KUKA KRL program: EPS_2_251078_MH1A_A_20250930064554.src

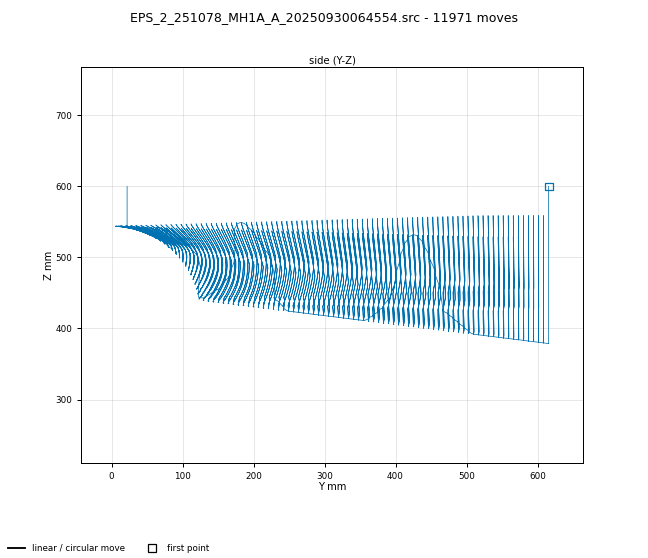
[picture p0: tool path of EPS_2_251078_MH1A_A_20250930064554.src, 11971 of 11973 moves have a stored position in this frame; points joined in program order, loops and branches not executed]
&ACCESS RVP
&REL 4
&COMMENT QRS 19112012
&PARAM EDITMASK = *
DEF PART()
EXT BAS (BAS_COMMAND :IN,REAL :IN )
INT I
BAS (#INITMOV,0 )

;KUKA QRS Post kuka4.cps  Date:22-06-2017 !

File_ID=2857

QRS_PRE_INIT()

;Init var - Until changes are made in qrs_pre_init
Outlet_Square_prg=0
Inlet_1_Square_prg=0
Inlet_2_Square_prg=0
Inlet_3_Square_prg=0
Inlet_4_Square_prg=0
Inlet_5_Square_prg=0

Outlet_1={X 0.000, Y 520.860, Z 458.500, B 0.000, E1 0.000 }
Inlet_1={X 0.000, Y 523.030, Z 428.500, B 0.000, E1 180.000 }
Outlet_1_type=201
Inlet_1_type=201
;QRS#1=Sidecore dimensions
;QRS#2=200-8" PVC SDR 35
;QRS#3=200-8" PVC SDR 35
;QRS#4=
;QRS#5=
;QRS#6=
;QRS#7=
;QRS#8=
;QRS#9=12-08 PSX
;QRS#10=12-08 PSX
;QRS#11=
;QRS#12=
;QRS#13=
;QRS#14=
;QRS#15=
;QRS#16=1220x127x838 2,75'
;QRS#17=EPS Height
;QRS#18=559
;QRS#19=*
;QRS#20= UPDATED VERSION 22-06-2017
;QRS#21=*
Outlet_Square=0100
Inlet_1_Square=0100
Inlet_2_Square=0
Inlet_3_Square=0
Inlet_4_Square=0
Inlet_5_Square=0
Mill_Square=1
Outlet_Square_Prg=204
Inlet_1_Square_prg=204

QRS_INIT()

$ADVANCE=5

; T1
PTP {E1 173.607,E2 173.607}
PTP {X 0,Y 615.504,A -85,B 0,C 180,E1 173.607,E2 173.607,E3 0,E4 0,E5 0,E6 0}
QRS_SPEED_INIT()
LIN {X 0,Y 615.504,Z 600,A -85,B 0,C 180,E1 173.607,E2 173.607,E3 0,E4 0,E5 0,E6 0} C_VEL
LIN {X 0,Y 615.504,Z 388.868,A -85,B 0,C 180,E1 173.607,E2 173.607} C_VEL
LIN {X 0,Y 615.504,Z 380.694,A -85,B 0,C 180,E1 173.607,E2 173.607} C_VEL
LIN {X 0,Y 615.49,Z 378.694,A -85,B 0,C 180,E1 173.421,E2 173.421} C_VEL
LIN {X 0,Y 615.492,Z 378.688,A -85,B 0,C 180,E1 170.801,E2 170.801} C_VEL
LIN {X 0,Y 615.493,Z 378.697,A -85,B 0,C 180,E1 168.139,E2 168.139} C_VEL
LIN {X 0,Y 615.481,Z 378.689,A -85,B 0,C 180,E1 165.451,E2 165.451} C_VEL
LIN {X 0,Y 615.492,Z 378.698,A -85,B 0,C 180,E1 162.73,E2 162.73} C_VEL
LIN {X 0,Y 615.49,Z 378.689,A -85,B 0,C 180,E1 159.967,E2 159.967} C_VEL
LIN {X 0,Y 615.486,Z 378.69,A -85,B 0,C 180,E1 157.155,E2 157.155} C_VEL
LIN {X 0,Y 615.5,Z 378.7,A -85,B 0,C 180,E1 154.285,E2 154.285} C_VEL
LIN {X 0,Y 615.478,Z 378.69,A -85,B 0,C 180,E1 151.552,E2 151.552} C_VEL
LIN {X 0,Y 615.487,Z 378.696,A -85,B 0,C 180,E1 148.914,E2 148.914} C_VEL
LIN {X 0,Y 615.489,Z 378.694,A -85,B 0,C 180,E1 145.978,E2 145.978} C_VEL
LIN {X 0,Y 615.487,Z 378.688,A -85,B 0,C 180,E1 143.064,E2 143.064} C_VEL
LIN {X 0,Y 615.49,Z 378.693,A -85,B 0,C 180,E1 140.25,E2 140.25} C_VEL
LIN {X 0,Y 615.477,Z 378.692,A -85,B 0,C 180,E1 137.646,E2 137.646} C_VEL
LIN {X 0,Y 615.48,Z 378.692,A -85,B 0,C 180,E1 134.93,E2 134.93} C_VEL
LIN {X 0,Y 615.49,Z 378.7,A -85,B 0,C 180,E1 132.08,E2 132.08} C_VEL
LIN {X 0,Y 615.479,Z 378.691,A -85,B 0,C 180,E1 129.751,E2 129.751} C_VEL
LIN {X 0,Y 615.488,Z 378.7,A -85,B 0,C 180,E1 126.936,E2 126.936} C_VEL
LIN {X 0,Y 615.485,Z 378.691,A -85,B 0,C 180,E1 125.616,E2 125.616} C_VEL
LIN {X 0,Y 615.482,Z 379.783,A -85,B 0,C 180,E1 124.699,E2 124.699} C_VEL
LIN {X 0,Y 615.494,Z 383.903,A -85,B 0,C 180,E1 122.331,E2 122.331} C_VEL
LIN {X 0,Y 615.496,Z 389.153,A -85,B 0,C 180,E1 119.406,E2 119.406} C_VEL
LIN {X 0,Y 615.486,Z 394.642,A -85,B 0,C 180,E1 116.444,E2 116.444} C_VEL
LIN {X 0,Y 615.49,Z 400.151,A -85,B 0,C 180,E1 113.556,E2 113.556} C_VEL
LIN {X 0,Y 615.487,Z 405.633,A -85,B 0,C 180,E1 110.731,E2 110.731} C_VEL
LIN {X 0,Y 615.483,Z 411.136,A -85,B 0,C 180,E1 107.957,E2 107.957} C_VEL
LIN {X 0,Y 615.484,Z 416.622,A -85,B 0,C 180,E1 105.226,E2 105.226} C_VEL
LIN {X 0,Y 615.483,Z 422.111,A -85,B 0,C 180,E1 102.53,E2 102.53} C_VEL
LIN {X 0,Y 615.492,Z 424.087,A -85,B 0,C 180,E1 101.568,E2 101.568} C_VEL
LIN {X 0,Y 615.484,Z 438.741,A -85,B 0,C 180,E1 101.235,E2 101.235} C_VEL
LIN {X 0,Y 615.491,Z 450.62,A -85,B 0,C 180,E1 100.842,E2 100.842} C_VEL
LIN {X 0,Y 615.478,Z 461.568,A -85,B 0,C 180,E1 100.361,E2 100.361} C_VEL
LIN {X 0,Y 615.497,Z 473.304,A -85,B 0,C 180,E1 99.696,E2 99.696} C_VEL
LIN {X 0,Y 615.499,Z 483.768,A -85,B 0,C 180,E1 98.95,E2 98.95} C_VEL
LIN {X 0,Y 615.498,Z 492.331,A -85,B 0,C 180,E1 98.206,E2 98.206} C_VEL
LIN {X 0,Y 615.497,Z 500.21,A -85,B 0,C 180,E1 97.38,E2 97.38} C_VEL
LIN {X 0,Y 615.497,Z 507.899,A -85,B 0,C 180,E1 96.392,E2 96.392} C_VEL
LIN {X 0,Y 615.497,Z 514.958,A -85,B 0,C 180,E1 95.241,E2 95.241} C_VEL
LIN {X 0,Y 615.494,Z 519.658,A -85,B 0,C 180,E1 94.256,E2 94.256} C_VEL
LIN {X 0,Y 615.494,Z 523.255,A -85,B 0,C 180,E1 93.273,E2 93.273} C_VEL
LIN {X 0,Y 615.496,Z 525.115,A -85,B 0,C 180,E1 92.618,E2 92.618} C_VEL
LIN {X 0,Y 615.5,Z 526.533,A -85,B 0,C 180,E1 91.963,E2 91.963} C_VEL
LIN {X 0,Y 615.496,Z 528.142,A -85,B 0,C 180,E1 90.654,E2 90.654} C_VEL
LIN {X 0,Y 615.495,Z 528.384,A -85,B 0,C 180,E1 90,E2 90} C_VEL
LIN {X 0,Y 615.495,Z 528.206,A -85,B 0,C 180,E1 89.346,E2 89.346} C_VEL
LIN {X 0,Y 615.5,Z 526.682,A -85,B 0,C 180,E1 88.037,E2 88.037} C_VEL
LIN {X 0,Y 615.498,Z 525.341,A -85,B 0,C 180,E1 87.382,E2 87.382} C_VEL
LIN {X 0,Y 615.496,Z 522.494,A -85,B 0,C 180,E1 86.399,E2 86.399} C_VEL
LIN {X 0,Y 615.498,Z 518.634,A -85,B 0,C 180,E1 85.415,E2 85.415} C_VEL
LIN {X 0,Y 615.498,Z 513.651,A -85,B 0,C 180,E1 84.43,E2 84.43} C_VEL
LIN {X 0,Y 615.496,Z 507.208,A -85,B 0,C 180,E1 83.418,E2 83.418} C_VEL
LIN {X 0,Y 615.497,Z 499.536,A -85,B 0,C 180,E1 82.455,E2 82.455} C_VEL
LIN {X 0,Y 615.498,Z 489.758,A -85,B 0,C 180,E1 81.463,E2 81.463} C_VEL
LIN {X 0,Y 615.498,Z 479.491,A -85,B 0,C 180,E1 80.636,E2 80.636} C_VEL
LIN {X 0,Y 615.482,Z 467.93,A -85,B 0,C 180,E1 79.889,E2 79.889} C_VEL
LIN {X 0,Y 615.491,Z 456.089,A -85,B 0,C 180,E1 79.294,E2 79.294} C_VEL
LIN {X 0,Y 615.477,Z 443.158,A -85,B 0,C 180,E1 78.807,E2 78.807} C_VEL
LIN {X 0,Y 615.487,Z 430.554,A -85,B 0,C 180,E1 78.473,E2 78.473} C_VEL
LIN {X 0,Y 615.496,Z 424.099,A -85,B 0,C 180,E1 78.348,E2 78.348} C_VEL
LIN {X 0,Y 615.481,Z 418.176,A -85,B 0,C 180,E1 75.451,E2 75.451} C_VEL
LIN {X 0,Y 615.486,Z 412.683,A -85,B 0,C 180,E1 72.729,E2 72.729} C_VEL
LIN {X 0,Y 615.479,Z 407.193,A -85,B 0,C 180,E1 69.967,E2 69.967} C_VEL
LIN {X 0,Y 615.486,Z 401.687,A -85,B 0,C 180,E1 67.155,E2 67.155} C_VEL
LIN {X 0,Y 615.487,Z 396.196,A -85,B 0,C 180,E1 64.284,E2 64.284} C_VEL
LIN {X 0,Y 615.491,Z 391.067,A -85,B 0,C 180,E1 61.55,E2 61.55} C_VEL
LIN {X 0,Y 615.488,Z 386.262,A -85,B 0,C 180,E1 58.914,E2 58.914} C_VEL
LIN {X 0,Y 615.495,Z 381.958,A -85,B 0,C 180,E1 56.465,E2 56.465} C_VEL
LIN {X 0,Y 615.483,Z 379.738,A -85,B 0,C 180,E1 55.184,E2 55.184} C_VEL
LIN {X 0,Y 615.485,Z 378.693,A -85,B 0,C 180,E1 54.384,E2 54.384} C_VEL
LIN {X 0,Y 615.481,Z 378.69,A -85,B 0,C 180,E1 51.931,E2 51.931} C_VEL
LIN {X 0,Y 615.485,Z 378.696,A -85,B 0,C 180,E1 49.393,E2 49.393} C_VEL
LIN {X 0,Y 615.496,Z 378.687,A -85,B 0,C 180,E1 46.756,E2 46.756} C_VEL
LIN {X 0,Y 615.484,Z 378.691,A -85,B 0,C 180,E1 43.997,E2 43.997} C_VEL
LIN {X 0,Y 615.491,Z 378.701,A -85,B 0,C 180,E1 41.095,E2 41.095} C_VEL
LIN {X 0,Y 615.494,Z 378.69,A -85,B 0,C 180,E1 38.904,E2 38.904} C_VEL
LIN {X 0,Y 615.478,Z 378.692,A -85,B 0,C 180,E1 36.426,E2 36.426} C_VEL
LIN {X 0,Y 615.487,Z 378.697,A -85,B 0,C 180,E1 34.022,E2 34.022} C_VEL
LIN {X 0,Y 615.482,Z 378.689,A -85,B 0,C 180,E1 31.686,E2 31.686} C_VEL
LIN {X 0,Y 615.48,Z 378.695,A -85,B 0,C 180,E1 29.407,E2 29.407} C_VEL
LIN {X 0,Y 615.498,Z 378.691,A -85,B 0,C 180,E1 27.046,E2 27.046} C_VEL
LIN {X 0,Y 615.487,Z 378.693,A -85,B 0,C 180,E1 24.272,E2 24.272} C_VEL
LIN {X 0,Y 615.479,Z 378.689,A -85,B 0,C 180,E1 21.432,E2 21.432} C_VEL
LIN {X 0,Y 615.481,Z 378.698,A -85,B 0,C 180,E1 18.602,E2 18.602} C_VEL
LIN {X 0,Y 615.48,Z 378.691,A -85,B 0,C 180,E1 15.905,E2 15.905} C_VEL
LIN {X 0,Y 615.494,Z 378.689,A -85,B 0,C 180,E1 13.201,E2 13.201} C_VEL
LIN {X 0,Y 615.486,Z 378.695,A -85,B 0,C 180,E1 10.527,E2 10.527} C_VEL
LIN {X 0,Y 615.477,Z 378.691,A -85,B 0,C 180,E1 7.876,E2 7.876} C_VEL
LIN {X 0,Y 615.495,Z 378.697,A -85,B 0,C 180,E1 5.241,E2 5.241} C_VEL
LIN {X 0,Y 615.488,Z 378.688,A -85,B 0,C 180,E1 2.618,E2 2.618} C_VEL
LIN {X 0,Y 615.486,Z 378.702,A -85,B 0,C 180,E1 0,E2 0} C_VEL
LIN {X 0,Y 615.488,Z 378.687,A -85,B 0,C 180,E1 -2.618,E2 -2.618} C_VEL
LIN {X 0,Y 615.489,Z 378.7,A -85,B 0,C 180,E1 -5.241,E2 -5.241} C_VEL
LIN {X 0,Y 615.478,Z 378.69,A -85,B 0,C 180,E1 -7.876,E2 -7.876} C_VEL
LIN {X 0,Y 615.485,Z 378.697,A -85,B 0,C 180,E1 -10.527,E2 -10.527} C_VEL
LIN {X 0,Y 615.494,Z 378.688,A -85,B 0,C 180,E1 -13.201,E2 -13.201} C_VEL
LIN {X 0,Y 615.485,Z 378.691,A -85,B 0,C 180,E1 -15.905,E2 -15.905} C_VEL
LIN {X 0,Y 615.49,Z 378.695,A -85,B 0,C 180,E1 -18.646,E2 -18.646} C_VEL
LIN {X 0,Y 615.478,Z 378.69,A -85,B 0,C 180,E1 -21.432,E2 -21.432} C_VEL
LIN {X 0,Y 615.484,Z 378.696,A -85,B 0,C 180,E1 -24.272,E2 -24.272} C_VEL
LIN {X 0,Y 615.497,Z 378.69,A -85,B 0,C 180,E1 -27.046,E2 -27.046} C_VEL
LIN {X 0,Y 615.488,Z 378.688,A -85,B 0,C 180,E1 -29.794,E2 -29.794} C_VEL
LIN {X 0,Y 615.49,Z 378.698,A -85,B 0,C 180,E1 -32.457,E2 -32.457} C_VEL
LIN {X 0,Y 615.49,Z 378.689,A -85,B 0,C 180,E1 -34.815,E2 -34.815} C_VEL
LIN {X 0,Y 615.481,Z 378.692,A -85,B 0,C 180,E1 -37.243,E2 -37.243} C_VEL
LIN {X 0,Y 615.483,Z 378.689,A -85,B 0,C 180,E1 -40.088,E2 -40.088} C_VEL
LIN {X 0,Y 615.477,Z 378.692,A -85,B 0,C 180,E1 -42.354,E2 -42.354} C_VEL
LIN {X 0,Y 615.48,Z 378.692,A -85,B 0,C 180,E1 -45.069,E2 -45.069} C_VEL
LIN {X 0,Y 615.495,Z 378.699,A -85,B 0,C 180,E1 -47.919,E2 -47.919} C_VEL
LIN {X 0,Y 615.478,Z 378.692,A -85,B 0,C 180,E1 -50.249,E2 -50.249} C_VEL
LIN {X 0,Y 615.483,Z 378.702,A -85,B 0,C 180,E1 -53.064,E2 -53.064} C_VEL
LIN {X 0,Y 615.49,Z 378.789,A -85,B 0,C 180,E1 -54.585,E2 -54.585} C_VEL
LIN {X 0,Y 615.495,Z 387.112,A -85,B 0,C 180,E1 -57.543,E2 -57.543} C_VEL
LIN {X 0,Y 615.479,Z 394.86,A -85,B 0,C 180,E1 -60.207,E2 -60.207} C_VEL
LIN {X 0,Y 615.478,Z 403.061,A -85,B 0,C 180,E1 -62.957,E2 -62.957} C_VEL
LIN {X 0,Y 615.495,Z 411.522,A -85,B 0,C 180,E1 -65.728,E2 -65.728} C_VEL
LIN {X 0,Y 615.485,Z 420.39,A -85,B 0,C 180,E1 -68.568,E2 -68.568} C_VEL
LIN {X 0,Y 615.488,Z 429.381,A -85,B 0,C 180,E1 -71.396,E2 -71.396} C_VEL
LIN {X 0,Y 615.485,Z 438.108,A -85,B 0,C 180,E1 -74.095,E2 -74.095} C_VEL
LIN {X 0,Y 615.494,Z 446.951,A -85,B 0,C 180,E1 -76.799,E2 -76.799} C_VEL
LIN {X 0,Y 615.491,Z 452.137,A -85,B 0,C 180,E1 -78.369,E2 -78.369} C_VEL
LIN {X 0,Y 615.499,Z 465.817,A -85,B 0,C 180,E1 -78.64,E2 -78.64} C_VEL
LIN {X 0,Y 615.489,Z 478.534,A -85,B 0,C 180,E1 -79.036,E2 -79.036} C_VEL
LIN {X 0,Y 615.479,Z 490.765,A -85,B 0,C 180,E1 -79.556,E2 -79.556} C_VEL
LIN {X 0,Y 615.498,Z 501.385,A -85,B 0,C 180,E1 -80.138,E2 -80.138} C_VEL
LIN {X 0,Y 615.498,Z 512.23,A -85,B 0,C 180,E1 -80.884,E2 -80.884} C_VEL
LIN {X 0,Y 615.497,Z 522.811,A -85,B 0,C 180,E1 -81.794,E2 -81.794} C_VEL
LIN {X 0,Y 615.498,Z 530.605,A -85,B 0,C 180,E1 -82.619,E2 -82.619} C_VEL
LIN {X 0,Y 615.496,Z 538.202,A -85,B 0,C 180,E1 -83.608,E2 -83.608} C_VEL
LIN {X 0,Y 615.498,Z 545.204,A -85,B 0,C 180,E1 -84.759,E2 -84.759} C_VEL
LIN {X 0,Y 615.493,Z 549.851,A -85,B 0,C 180,E1 -85.744,E2 -85.744} C_VEL
LIN {X 0,Y 615.495,Z 553.398,A -85,B 0,C 180,E1 -86.727,E2 -86.727} C_VEL
LIN {X 0,Y 615.497,Z 555.233,A -85,B 0,C 180,E1 -87.382,E2 -87.382} C_VEL
LIN {X 0,Y 615.499,Z 556.607,A -85,B 0,C 180,E1 -88.037,E2 -88.037} C_VEL
LIN {X 0,Y 615.496,Z 558.173,A -85,B 0,C 180,E1 -89.346,E2 -89.346} C_VEL
LIN {X 0,Y 615.494,Z 558.389,A -85,B 0,C 180,E1 -90,E2 -90} C_VEL
LIN {X 0,Y 615.496,Z 557.58,A -85,B 0,C 180,E1 -91.309,E2 -91.309} C_VEL
LIN {X 0,Y 615.499,Z 556.608,A -85,B 0,C 180,E1 -91.963,E2 -91.963} C_VEL
LIN {X 0,Y 615.497,Z 555.233,A -85,B 0,C 180,E1 -92.618,E2 -92.618} C_VEL
LIN {X 0,Y 615.496,Z 552.35,A -85,B 0,C 180,E1 -93.601,E2 -93.601} C_VEL
LIN {X 0,Y 615.498,Z 548.442,A -85,B 0,C 180,E1 -94.584,E2 -94.584} C_VEL
LIN {X 0,Y 615.499,Z 543.405,A -85,B 0,C 180,E1 -95.57,E2 -95.57} C_VEL
LIN {X 0,Y 615.497,Z 536.869,A -85,B 0,C 180,E1 -96.583,E2 -96.583} C_VEL
LIN {X 0,Y 615.497,Z 529.133,A -85,B 0,C 180,E1 -97.545,E2 -97.545} C_VEL
LIN {X 0,Y 615.498,Z 521.045,A -85,B 0,C 180,E1 -98.371,E2 -98.371} C_VEL
LIN {X 0,Y 615.499,Z 511.168,A -85,B 0,C 180,E1 -99.199,E2 -99.199} C_VEL
LIN {X 0,Y 615.491,Z 499.981,A -85,B 0,C 180,E1 -99.945,E2 -99.945} C_VEL
LIN {X 0,Y 615.481,Z 489.024,A -85,B 0,C 180,E1 -100.527,E2 -100.527} C_VEL
LIN {X 0,Y 615.489,Z 476.47,A -85,B 0,C 180,E1 -101.041,E2 -101.041} C_VEL
LIN {X 0,Y 615.498,Z 464.064,A -85,B 0,C 180,E1 -101.401,E2 -101.401} C_VEL
LIN {X 0,Y 615.491,Z 452.138,A -85,B 0,C 180,E1 -101.631,E2 -101.631} C_VEL
LIN {X 0,Y 615.476,Z 443.545,A -85,B 0,C 180,E1 -104.24,E2 -104.24} C_VEL
LIN {X 0,Y 615.483,Z 434.783,A -85,B 0,C 180,E1 -106.928,E2 -106.928} C_VEL
LIN {X 0,Y 615.485,Z 425.928,A -85,B 0,C 180,E1 -109.685,E2 -109.685} C_VEL
LIN {X 0,Y 615.491,Z 417.513,A -85,B 0,C 180,E1 -112.346,E2 -112.346} C_VEL
LIN {X 0,Y 615.478,Z 409.309,A -85,B 0,C 180,E1 -114.992,E2 -114.992} C_VEL
LIN {X 0,Y 615.494,Z 401.542,A -85,B 0,C 180,E1 -117.545,E2 -117.545} C_VEL
LIN {X 0,Y 615.497,Z 392.668,A -85,B 0,C 180,E1 -120.539,E2 -120.539} C_VEL
LIN {X 0,Y 615.491,Z 384.883,A -85,B 0,C 180,E1 -123.236,E2 -123.236} C_VEL
LIN {X 0,Y 615.489,Z 378.692,A -85,B 0,C 180,E1 -125.515,E2 -125.515} C_VEL
LIN {X 0,Y 615.481,Z 378.691,A -85,B 0,C 180,E1 -128.069,E2 -128.069} C_VEL
LIN {X 0,Y 615.482,Z 378.695,A -85,B 0,C 180,E1 -130.607,E2 -130.607} C_VEL
LIN {X 0,Y 615.496,Z 378.688,A -85,B 0,C 180,E1 -133.244,E2 -133.244} C_VEL
LIN {X 0,Y 615.488,Z 378.689,A -85,B 0,C 180,E1 -136.003,E2 -136.003} C_VEL
LIN {X 0,Y 615.488,Z 378.702,A -85,B 0,C 180,E1 -138.906,E2 -138.906} C_VEL
LIN {X 0,Y 615.49,Z 378.689,A -85,B 0,C 180,E1 -141.096,E2 -141.096} C_VEL
LIN {X 0,Y 615.478,Z 378.693,A -85,B 0,C 180,E1 -143.574,E2 -143.574} C_VEL
LIN {X 0,Y 615.494,Z 378.694,A -85,B 0,C 180,E1 -145.978,E2 -145.978} C_VEL
LIN {X 0,Y 615.482,Z 378.689,A -85,B 0,C 180,E1 -148.314,E2 -148.314} C_VEL
LIN {X 0,Y 615.483,Z 378.696,A -85,B 0,C 180,E1 -150.593,E2 -150.593} C_VEL
LIN {X 0,Y 615.497,Z 378.69,A -85,B 0,C 180,E1 -152.953,E2 -152.953} C_VEL
LIN {X 0,Y 615.484,Z 378.695,A -85,B 0,C 180,E1 -155.728,E2 -155.728} C_VEL
LIN {X 0,Y 615.478,Z 378.689,A -85,B 0,C 180,E1 -158.568,E2 -158.568} C_VEL
LIN {X 0,Y 615.488,Z 378.695,A -85,B 0,C 180,E1 -161.396,E2 -161.396} C_VEL
LIN {X 0,Y 615.482,Z 378.692,A -85,B 0,C 180,E1 -164.095,E2 -164.095} C_VEL
LIN {X 0,Y 615.494,Z 378.689,A -85,B 0,C 180,E1 -166.799,E2 -166.799} C_VEL
LIN {X 0,Y 615.486,Z 378.696,A -85,B 0,C 180,E1 -169.473,E2 -169.473} C_VEL
LIN {X 0,Y 615.478,Z 378.69,A -85,B 0,C 180,E1 -172.124,E2 -172.124} C_VEL
LIN {X 0,Y 615.489,Z 378.699,A -85,B 0,C 180,E1 -174.759,E2 -174.759} C_VEL
LIN {X 0,Y 615.488,Z 378.687,A -85,B 0,C 180,E1 -177.382,E2 -177.382} C_VEL
LIN {X 0,Y 615.489,Z 378.702,A -85,B 0,C 180,E1 -180,E2 -180} C_VEL
LIN {X 0,Y 615.488,Z 378.687,A -85,B 0,C 180,E1 -182.618,E2 -182.618} C_VEL
LIN {X 0,Y 615.495,Z 378.698,A -85,B 0,C 180,E1 -185.241,E2 -185.241} C_VEL
LIN {X 0,Y 615.49,Z 378.694,A -85,B 0,C 180,E1 -186.579,E2 -186.579} C_VEL
LIN {X 0,Y 614.817,Z 378.84,A -85,B 0,C 180,E1 -187.125,E2 -187.125} C_VEL
LIN {X 0,Y 611.985,Z 379.251,A -85,B 0,C 180,E1 -188.011,E2 -188.011} C_VEL
LIN {X 0,Y 609.592,Z 379.56,A -85,B 0,C 180,E1 -188.724,E2 -188.724} C_VEL
LIN {X 0,Y 608.552,Z 379.679,A -85,B 0,C 180,E1 -189.273,E2 -189.273} C_VEL
LIN {X 0,Y 608.461,Z 379.689,A -85,B 0,C 180,E1 -189.459,E2 -189.459} C_VEL
LIN {X 0,Y 608.466,Z 379.697,A -85,B 0,C 180,E1 -192,E2 -192} C_VEL
LIN {X 0,Y 608.474,Z 379.688,A -85,B 0,C 180,E1 -194.721,E2 -194.721} C_VEL
LIN {X 0,Y 608.455,Z 379.693,A -85,B 0,C 180,E1 -197.477,E2 -197.477} C_VEL
LIN {X 0,Y 608.465,Z 379.692,A -85,B 0,C 180,E1 -200.274,E2 -200.274} C_VEL
LIN {X 0,Y 608.449,Z 379.691,A -85,B 0,C 180,E1 -203.124,E2 -203.124} C_VEL
LIN {X 0,Y 608.481,Z 379.695,A -85,B 0,C 180,E1 -205.722,E2 -205.722} C_VEL
LIN {X 0,Y 608.446,Z 379.691,A -85,B 0,C 180,E1 -208.267,E2 -208.267} C_VEL
LIN {X 0,Y 608.476,Z 379.69,A -85,B 0,C 180,E1 -210.545,E2 -210.545} C_VEL
LIN {X 0,Y 608.455,Z 379.693,A -85,B 0,C 180,E1 -212.88,E2 -212.88} C_VEL
LIN {X 0,Y 608.443,Z 379.691,A -85,B 0,C 180,E1 -215.278,E2 -215.278} C_VEL
LIN {X 0,Y 608.468,Z 379.696,A -85,B 0,C 180,E1 -217.747,E2 -217.747} C_VEL
LIN {X 0,Y 608.448,Z 379.691,A -85,B 0,C 180,E1 -220.328,E2 -220.328} C_VEL
LIN {X 0,Y 608.449,Z 379.697,A -85,B 0,C 180,E1 -222.96,E2 -222.96} C_VEL
LIN {X 0,Y 608.46,Z 379.69,A -85,B 0,C 180,E1 -225.736,E2 -225.736} C_VEL
LIN {X 0,Y 608.465,Z 379.689,A -85,B 0,C 180,E1 -228.658,E2 -228.658} C_VEL
LIN {X 0,Y 608.465,Z 379.692,A -85,B 0,C 180,E1 -231.76,E2 -231.76} C_VEL
LIN {X 0,Y 608.447,Z 379.691,A -85,B 0,C 180,E1 -233.955,E2 -233.955} C_VEL
LIN {X 0,Y 608.413,Z 379.769,A -85,B 0,C 180,E1 -234.72,E2 -234.72} C_VEL
LIN {X 0,Y 608.464,Z 383.894,A -85,B 0,C 180,E1 -237.121,E2 -237.121} C_VEL
LIN {X 0,Y 608.443,Z 389.024,A -85,B 0,C 180,E1 -240.033,E2 -240.033} C_VEL
LIN {X 0,Y 608.445,Z 394.097,A -85,B 0,C 180,E1 -242.799,E2 -242.799} C_VEL
LIN {X 0,Y 608.423,Z 399.036,A -85,B 0,C 180,E1 -245.428,E2 -245.428} C_VEL
LIN {X 0,Y 608.446,Z 404.566,A -85,B 0,C 180,E1 -248.308,E2 -248.308} C_VEL
LIN {X 0,Y 608.427,Z 410.427,A -85,B 0,C 180,E1 -251.297,E2 -251.297} C_VEL
LIN {X 0,Y 608.442,Z 415.625,A -85,B 0,C 180,E1 -253.906,E2 -253.906} C_VEL
LIN {X 0,Y 608.425,Z 421.155,A -85,B 0,C 180,E1 -256.643,E2 -256.643} C_VEL
LIN {X 0,Y 608.45,Z 424.524,A -85,B 0,C 180,E1 -258.296,E2 -258.296} C_VEL
LIN {X 0,Y 608.526,Z 440.394,A -85,B 0,C 180,E1 -258.677,E2 -258.677} C_VEL
LIN {X 0,Y 608.532,Z 452.792,A -85,B 0,C 180,E1 -259.113,E2 -259.113} C_VEL
LIN {X 0,Y 608.48,Z 464.935,A -85,B 0,C 180,E1 -259.687,E2 -259.687} C_VEL
LIN {X 0,Y 608.5,Z 476.067,A -85,B 0,C 180,E1 -260.359,E2 -260.359} C_VEL
LIN {X 0,Y 608.474,Z 485.084,A -85,B 0,C 180,E1 -261.029,E2 -261.029} C_VEL
LIN {X 0,Y 608.464,Z 494.35,A -85,B 0,C 180,E1 -261.866,E2 -261.866} C_VEL
LIN {X 0,Y 608.466,Z 503.324,A -85,B 0,C 180,E1 -262.867,E2 -262.867} C_VEL
LIN {X 0,Y 608.444,Z 510.556,A -85,B 0,C 180,E1 -263.867,E2 -263.867} C_VEL
LIN {X 0,Y 608.462,Z 515.435,A -85,B 0,C 180,E1 -264.698,E2 -264.698} C_VEL
LIN {X 0,Y 608.439,Z 520.178,A -85,B 0,C 180,E1 -265.694,E2 -265.694} C_VEL
LIN {X 0,Y 608.425,Z 523.812,A -85,B 0,C 180,E1 -266.689,E2 -266.689} C_VEL
LIN {X 0,Y 608.425,Z 525.691,A -85,B 0,C 180,E1 -267.352,E2 -267.352} C_VEL
LIN {X 0,Y 608.444,Z 527.127,A -85,B 0,C 180,E1 -268.014,E2 -268.014} C_VEL
LIN {X 0,Y 608.439,Z 528.752,A -85,B 0,C 180,E1 -269.338,E2 -269.338} C_VEL
LIN {X 0,Y 608.435,Z 528.995,A -85,B 0,C 180,E1 -270,E2 -270} C_VEL
LIN {X 0,Y 608.438,Z 528.815,A -85,B 0,C 180,E1 -270.662,E2 -270.662} C_VEL
LIN {X 0,Y 608.445,Z 527.276,A -85,B 0,C 180,E1 -271.986,E2 -271.986} C_VEL
LIN {X 0,Y 608.426,Z 525.918,A -85,B 0,C 180,E1 -272.648,E2 -272.648} C_VEL
LIN {X 0,Y 608.449,Z 523.041,A -85,B 0,C 180,E1 -273.642,E2 -273.642} C_VEL
LIN {X 0,Y 608.433,Z 519.142,A -85,B 0,C 180,E1 -274.638,E2 -274.638} C_VEL
LIN {X 0,Y 608.45,Z 514.112,A -85,B 0,C 180,E1 -275.634,E2 -275.634} C_VEL
LIN {X 0,Y 608.441,Z 507.794,A -85,B 0,C 180,E1 -276.633,E2 -276.633} C_VEL
LIN {X 0,Y 608.475,Z 499.878,A -85,B 0,C 180,E1 -277.633,E2 -277.633} C_VEL
LIN {X 0,Y 608.472,Z 490.035,A -85,B 0,C 180,E1 -278.636,E2 -278.636} C_VEL
LIN {X 0,Y 608.481,Z 479.712,A -85,B 0,C 180,E1 -279.473,E2 -279.473} C_VEL
LIN {X 0,Y 608.478,Z 468.098,A -85,B 0,C 180,E1 -280.229,E2 -280.229} C_VEL
LIN {X 0,Y 608.507,Z 456.22,A -85,B 0,C 180,E1 -280.831,E2 -280.831} C_VEL
LIN {X 0,Y 608.521,Z 443.258,A -85,B 0,C 180,E1 -281.323,E2 -281.323} C_VEL
LIN {X 0,Y 608.546,Z 430.64,A -85,B 0,C 180,E1 -281.66,E2 -281.66} C_VEL
LIN {X 0,Y 608.446,Z 424.535,A -85,B 0,C 180,E1 -281.789,E2 -281.789} C_VEL
LIN {X 0,Y 608.413,Z 418.571,A -85,B 0,C 180,E1 -284.722,E2 -284.722} C_VEL
LIN {X 0,Y 608.432,Z 413.039,A -85,B 0,C 180,E1 -287.477,E2 -287.477} C_VEL
LIN {X 0,Y 608.425,Z 407.506,A -85,B 0,C 180,E1 -290.276,E2 -290.276} C_VEL
LIN {X 0,Y 608.432,Z 403.236,A -85,B 0,C 180,E1 -292.469,E2 -292.469} C_VEL
LIN {X 0,Y 608.435,Z 397.824,A -85,B 0,C 180,E1 -295.302,E2 -295.302} C_VEL
LIN {X 0,Y 608.45,Z 393.674,A -85,B 0,C 180,E1 -297.518,E2 -297.518} C_VEL
LIN {X 0,Y 608.443,Z 389.187,A -85,B 0,C 180,E1 -299.967,E2 -299.967} C_VEL
LIN {X 0,Y 608.465,Z 384.028,A -85,B 0,C 180,E1 -302.879,E2 -302.879} C_VEL
LIN {X 0,Y 608.414,Z 379.924,A -85,B 0,C 180,E1 -305.28,E2 -305.28} C_VEL
LIN {X 0,Y 608.484,Z 379.691,A -85,B 0,C 180,E1 -307.16,E2 -307.16} C_VEL
LIN {X 0,Y 608.443,Z 379.691,A -85,B 0,C 180,E1 -309.442,E2 -309.442} C_VEL
LIN {X 0,Y 608.466,Z 379.693,A -85,B 0,C 180,E1 -312.334,E2 -312.334} C_VEL
LIN {X 0,Y 608.452,Z 379.69,A -85,B 0,C 180,E1 -314.797,E2 -314.797} C_VEL
LIN {X 0,Y 608.448,Z 379.696,A -85,B 0,C 180,E1 -317.039,E2 -317.039} C_VEL
LIN {X 0,Y 608.456,Z 379.69,A -85,B 0,C 180,E1 -319.697,E2 -319.697} C_VEL
LIN {X 0,Y 608.467,Z 379.695,A -85,B 0,C 180,E1 -322.253,E2 -322.253} C_VEL
LIN {X 0,Y 608.456,Z 379.69,A -85,B 0,C 180,E1 -325.094,E2 -325.094} C_VEL
LIN {X 0,Y 608.465,Z 379.691,A -85,B 0,C 180,E1 -327.905,E2 -327.905} C_VEL
LIN {X 0,Y 608.47,Z 379.688,A -85,B 0,C 180,E1 -330.22,E2 -330.22} C_VEL
LIN {X 0,Y 608.488,Z 379.691,A -85,B 0,C 180,E1 -332.791,E2 -332.791} C_VEL
LIN {X 0,Y 608.457,Z 379.69,A -85,B 0,C 180,E1 -335.429,E2 -335.429} C_VEL
LIN {X 0,Y 608.468,Z 379.689,A -85,B 0,C 180,E1 -338.308,E2 -338.308} C_VEL
LIN {X 0,Y 608.457,Z 379.697,A -85,B 0,C 180,E1 -341.13,E2 -341.13} C_VEL
LIN {X 0,Y 608.458,Z 379.69,A -85,B 0,C 180,E1 -343.906,E2 -343.906} C_VEL
LIN {X 0,Y 608.468,Z 379.692,A -85,B 0,C 180,E1 -346.644,E2 -346.644} C_VEL
LIN {X 0,Y 608.462,Z 379.691,A -85,B 0,C 180,E1 -349.35,E2 -349.35} C_VEL
LIN {X 0,Y 608.473,Z 379.689,A -85,B 0,C 180,E1 -352.033,E2 -352.033} C_VEL
LIN {X 0,Y 608.472,Z 379.693,A -85,B 0,C 180,E1 -354.698,E2 -354.698} C_VEL
LIN {X 0,Y 608.479,Z 379.687,A -85,B 0,C 180,E1 -357.352,E2 -357.352} C_VEL
LIN {X 0,Y 608.477,Z 379.695,A -85,B 0,C 180,E1 -360,E2 -360} C_VEL
LIN {X 0,Y 608.479,Z 379.687,A -85,B 0,C 180,E1 -362.648,E2 -362.648} C_VEL
LIN {X 0,Y 608.467,Z 379.694,A -85,B 0,C 180,E1 -365.302,E2 -365.302} C_VEL
LIN {X 0,Y 608.473,Z 379.688,A -85,B 0,C 180,E1 -367.967,E2 -367.967} C_VEL
LIN {X 0,Y 608.461,Z 379.692,A -85,B 0,C 180,E1 -370.65,E2 -370.65} C_VEL
LIN {X 0,Y 608.471,Z 379.69,A -85,B 0,C 180,E1 -373.356,E2 -373.356} C_VEL
LIN {X 0,Y 608.461,Z 379.69,A -85,B 0,C 180,E1 -376.094,E2 -376.094} C_VEL
LIN {X 0,Y 608.46,Z 379.697,A -85,B 0,C 180,E1 -378.87,E2 -378.87} C_VEL
LIN {X 0,Y 608.467,Z 379.689,A -85,B 0,C 180,E1 -381.692,E2 -381.692} C_VEL
LIN {X 0,Y 608.455,Z 379.691,A -85,B 0,C 180,E1 -384.571,E2 -384.571} C_VEL
LIN {X 0,Y 608.488,Z 379.69,A -85,B 0,C 180,E1 -387.208,E2 -387.208} C_VEL
LIN {X 0,Y 608.47,Z 379.688,A -85,B 0,C 180,E1 -389.971,E2 -389.971} C_VEL
LIN {X 0,Y 608.458,Z 379.693,A -85,B 0,C 180,E1 -392.88,E2 -392.88} C_VEL
LIN {X 0,Y 608.442,Z 379.692,A -85,B 0,C 180,E1 -395.278,E2 -395.278} C_VEL
LIN {X 0,Y 608.467,Z 379.696,A -85,B 0,C 180,E1 -397.747,E2 -397.747} C_VEL
LIN {X 0,Y 608.447,Z 379.691,A -85,B 0,C 180,E1 -400.328,E2 -400.328} C_VEL
LIN {X 0,Y 608.452,Z 379.697,A -85,B 0,C 180,E1 -402.96,E2 -402.96} C_VEL
LIN {X 0,Y 608.463,Z 379.69,A -85,B 0,C 180,E1 -405.736,E2 -405.736} C_VEL
LIN {X 0,Y 608.463,Z 379.689,A -85,B 0,C 180,E1 -408.658,E2 -408.658} C_VEL
LIN {X 0,Y 608.464,Z 379.692,A -85,B 0,C 180,E1 -411.76,E2 -411.76} C_VEL
LIN {X 0,Y 608.513,Z 379.891,A -85,B 0,C 180,E1 -414.524,E2 -414.524} C_VEL
LIN {X 0,Y 608.496,Z 388.146,A -85,B 0,C 180,E1 -417.473,E2 -417.473} C_VEL
LIN {X 0,Y 608.471,Z 396.073,A -85,B 0,C 180,E1 -420.22,E2 -420.22} C_VEL
LIN {X 0,Y 608.474,Z 403.68,A -85,B 0,C 180,E1 -422.794,E2 -422.794} C_VEL
LIN {X 0,Y 608.466,Z 411.656,A -85,B 0,C 180,E1 -425.429,E2 -425.429} C_VEL
LIN {X 0,Y 608.453,Z 420.56,A -85,B 0,C 180,E1 -428.308,E2 -428.308} C_VEL
LIN {X 0,Y 608.46,Z 429.465,A -85,B 0,C 180,E1 -431.13,E2 -431.13} C_VEL
LIN {X 0,Y 608.442,Z 438.369,A -85,B 0,C 180,E1 -433.906,E2 -433.906} C_VEL
LIN {X 0,Y 608.438,Z 447.274,A -85,B 0,C 180,E1 -436.643,E2 -436.643} C_VEL
LIN {X 0,Y 608.436,Z 452.491,A -85,B 0,C 180,E1 -438.232,E2 -438.232} C_VEL
LIN {X 0,Y 608.544,Z 466.693,A -85,B 0,C 180,E1 -438.53,E2 -438.53} C_VEL
LIN {X 0,Y 608.521,Z 479.464,A -85,B 0,C 180,E1 -438.939,E2 -438.939} C_VEL
LIN {X 0,Y 608.51,Z 490.919,A -85,B 0,C 180,E1 -439.435,E2 -439.435} C_VEL
LIN {X 0,Y 608.489,Z 501.577,A -85,B 0,C 180,E1 -440.023,E2 -440.023} C_VEL
LIN {X 0,Y 608.483,Z 512.473,A -85,B 0,C 180,E1 -440.778,E2 -440.778} C_VEL
LIN {X 0,Y 608.475,Z 523.111,A -85,B 0,C 180,E1 -441.699,E2 -441.699} C_VEL
LIN {X 0,Y 608.471,Z 530.959,A -85,B 0,C 180,E1 -442.534,E2 -442.534} C_VEL
LIN {X 0,Y 608.461,Z 538.286,A -85,B 0,C 180,E1 -443.484,E2 -443.484} C_VEL
LIN {X 0,Y 608.45,Z 543.865,A -85,B 0,C 180,E1 -444.366,E2 -444.366} C_VEL
LIN {X 0,Y 608.432,Z 548.95,A -85,B 0,C 180,E1 -445.362,E2 -445.362} C_VEL
LIN {X 0,Y 608.449,Z 552.896,A -85,B 0,C 180,E1 -446.358,E2 -446.358} C_VEL
LIN {X 0,Y 608.425,Z 555.809,A -85,B 0,C 180,E1 -447.352,E2 -447.352} C_VEL
LIN {X 0,Y 608.444,Z 557.201,A -85,B 0,C 180,E1 -448.014,E2 -448.014} C_VEL
LIN {X 0,Y 608.438,Z 558.783,A -85,B 0,C 180,E1 -449.338,E2 -449.338} C_VEL
LIN {X 0,Y 608.434,Z 559,A -85,B 0,C 180,E1 -450,E2 -450} C_VEL
LIN {X 0,Y 608.448,Z 558.184,A -85,B 0,C 180,E1 -451.324,E2 -451.324} C_VEL
LIN {X 0,Y 608.444,Z 557.201,A -85,B 0,C 180,E1 -451.986,E2 -451.986} C_VEL
LIN {X 0,Y 608.425,Z 555.809,A -85,B 0,C 180,E1 -452.648,E2 -452.648} C_VEL
LIN {X 0,Y 608.449,Z 552.896,A -85,B 0,C 180,E1 -453.642,E2 -453.642} C_VEL
LIN {X 0,Y 608.432,Z 548.95,A -85,B 0,C 180,E1 -454.638,E2 -454.638} C_VEL
LIN {X 0,Y 608.437,Z 542.877,A -85,B 0,C 180,E1 -455.801,E2 -455.801} C_VEL
LIN {X 0,Y 608.462,Z 536.235,A -85,B 0,C 180,E1 -456.799,E2 -456.799} C_VEL
LIN {X 0,Y 608.455,Z 527.989,A -85,B 0,C 180,E1 -457.8,E2 -457.8} C_VEL
LIN {X 0,Y 608.472,Z 519.537,A -85,B 0,C 180,E1 -458.636,E2 -458.636} C_VEL
LIN {X 0,Y 608.481,Z 509.091,A -85,B 0,C 180,E1 -459.473,E2 -459.473} C_VEL
LIN {X 0,Y 608.491,Z 498.756,A -85,B 0,C 180,E1 -460.145,E2 -460.145} C_VEL
LIN {X 0,Y 608.518,Z 487.26,A -85,B 0,C 180,E1 -460.74,E2 -460.74} C_VEL
LIN {X 0,Y 608.537,Z 474.892,A -85,B 0,C 180,E1 -461.224,E2 -461.224} C_VEL
LIN {X 0,Y 608.546,Z 461.44,A -85,B 0,C 180,E1 -461.597,E2 -461.597} C_VEL
LIN {X 0,Y 608.436,Z 452.492,A -85,B 0,C 180,E1 -461.768,E2 -461.768} C_VEL
LIN {X 0,Y 608.424,Z 443.935,A -85,B 0,C 180,E1 -464.38,E2 -464.38} C_VEL
LIN {X 0,Y 608.451,Z 436.144,A -85,B 0,C 180,E1 -466.784,E2 -466.784} C_VEL
LIN {X 0,Y 608.457,Z 427.239,A -85,B 0,C 180,E1 -469.57,E2 -469.57} C_VEL
LIN {X 0,Y 608.48,Z 418.335,A -85,B 0,C 180,E1 -472.405,E2 -472.405} C_VEL
LIN {X 0,Y 608.465,Z 410.543,A -85,B 0,C 180,E1 -474.935,E2 -474.935} C_VEL
LIN {X 0,Y 608.473,Z 402.752,A -85,B 0,C 180,E1 -477.517,E2 -477.517} C_VEL
LIN {X 0,Y 608.485,Z 395.504,A -85,B 0,C 180,E1 -479.974,E2 -479.974} C_VEL
LIN {X 0,Y 608.498,Z 387.146,A -85,B 0,C 180,E1 -482.877,E2 -482.877} C_VEL
LIN {X 0,Y 608.463,Z 379.692,A -85,B 0,C 180,E1 -485.581,E2 -485.581} C_VEL
LIN {X 0,Y 608.464,Z 379.692,A -85,B 0,C 180,E1 -488.24,E2 -488.24} C_VEL
LIN {X 0,Y 608.463,Z 379.689,A -85,B 0,C 180,E1 -491.342,E2 -491.342} C_VEL
LIN {X 0,Y 608.463,Z 379.69,A -85,B 0,C 180,E1 -494.264,E2 -494.264} C_VEL
LIN {X 0,Y 608.449,Z 379.697,A -85,B 0,C 180,E1 -497.04,E2 -497.04} C_VEL
LIN {X 0,Y 608.454,Z 379.69,A -85,B 0,C 180,E1 -499.697,E2 -499.697} C_VEL
LIN {X 0,Y 608.466,Z 379.696,A -85,B 0,C 180,E1 -502.253,E2 -502.253} C_VEL
LIN {X 0,Y 608.442,Z 379.692,A -85,B 0,C 180,E1 -504.722,E2 -504.722} C_VEL
LIN {X 0,Y 608.466,Z 379.696,A -85,B 0,C 180,E1 -507.477,E2 -507.477} C_VEL
LIN {X 0,Y 608.472,Z 379.688,A -85,B 0,C 180,E1 -510.221,E2 -510.221} C_VEL
LIN {X 0,Y 608.488,Z 379.69,A -85,B 0,C 180,E1 -512.791,E2 -512.791} C_VEL
LIN {X 0,Y 608.455,Z 379.691,A -85,B 0,C 180,E1 -515.429,E2 -515.429} C_VEL
LIN {X 0,Y 608.467,Z 379.689,A -85,B 0,C 180,E1 -518.308,E2 -518.308} C_VEL
LIN {X 0,Y 608.458,Z 379.697,A -85,B 0,C 180,E1 -521.13,E2 -521.13} C_VEL
LIN {X 0,Y 608.459,Z 379.69,A -85,B 0,C 180,E1 -523.906,E2 -523.906} C_VEL
LIN {X 0,Y 608.471,Z 379.691,A -85,B 0,C 180,E1 -526.644,E2 -526.644} C_VEL
LIN {X 0,Y 608.462,Z 379.692,A -85,B 0,C 180,E1 -529.35,E2 -529.35} C_VEL
LIN {X 0,Y 608.473,Z 379.688,A -85,B 0,C 180,E1 -532.033,E2 -532.033} C_VEL
LIN {X 0,Y 608.467,Z 379.694,A -85,B 0,C 180,E1 -534.698,E2 -534.698} C_VEL
LIN {X 0,Y 608.479,Z 379.687,A -85,B 0,C 180,E1 -537.352,E2 -537.352} C_VEL
LIN {X 0,Y 608.48,Z 379.695,A -85,B 0,C 180,E1 -540,E2 -540} C_VEL
LIN {X 0,Y 608.479,Z 379.687,A -85,B 0,C 180,E1 -542.648,E2 -542.648} C_VEL
LIN {X 0,Y 608.473,Z 379.693,A -85,B 0,C 180,E1 -545.302,E2 -545.302} C_VEL
LIN {X 0,Y 608.473,Z 379.688,A -85,B 0,C 180,E1 -547.967,E2 -547.967} C_VEL
LIN {X 0,Y 608.461,Z 379.689,A -85,B 0,C 180,E1 -549.459,E2 -549.459} C_VEL
LIN {X 0,Y 607.777,Z 379.779,A -85,B 0,C 180,E1 -550.012,E2 -550.012} C_VEL
LIN {X 0,Y 604.924,Z 380.136,A -85,B 0,C 180,E1 -550.909,E2 -550.909} C_VEL
LIN {X 0,Y 602.525,Z 380.436,A -85,B 0,C 180,E1 -551.63,E2 -551.63} C_VEL
LIN {X 0,Y 601.496,Z 380.562,A -85,B 0,C 180,E1 -552.187,E2 -552.187} C_VEL
LIN {X 0,Y 601.412,Z 380.57,A -85,B 0,C 180,E1 -552.376,E2 -552.376} C_VEL
LIN {X 0,Y 601.43,Z 380.566,A -85,B 0,C 180,E1 -554.897,E2 -554.897} C_VEL
LIN {X 0,Y 601.424,Z 380.571,A -85,B 0,C 180,E1 -556.986,E2 -556.986} C_VEL
LIN {X 0,Y 601.409,Z 380.568,A -85,B 0,C 180,E1 -559.809,E2 -559.809} C_VEL
LIN {X 0,Y 601.414,Z 380.569,A -85,B 0,C 180,E1 -562.683,E2 -562.683} C_VEL
LIN {X 0,Y 601.407,Z 380.568,A -85,B 0,C 180,E1 -564.879,E2 -564.879} C_VEL
LIN {X 0,Y 601.425,Z 380.573,A -85,B 0,C 180,E1 -567.364,E2 -567.364} C_VEL
LIN {X 0,Y 601.431,Z 380.565,A -85,B 0,C 180,E1 -570.164,E2 -570.164} C_VEL
LIN {X 0,Y 601.42,Z 380.572,A -85,B 0,C 180,E1 -572.715,E2 -572.715} C_VEL
LIN {X 0,Y 601.414,Z 380.567,A -85,B 0,C 180,E1 -575.114,E2 -575.114} C_VEL
LIN {X 0,Y 601.437,Z 380.568,A -85,B 0,C 180,E1 -577.419,E2 -577.419} C_VEL
LIN {X 0,Y 601.414,Z 380.568,A -85,B 0,C 180,E1 -579.995,E2 -579.995} C_VEL
LIN {X 0,Y 601.41,Z 380.573,A -85,B 0,C 180,E1 -582.671,E2 -582.671} C_VEL
LIN {X 0,Y 601.429,Z 380.565,A -85,B 0,C 180,E1 -585.482,E2 -585.482} C_VEL
LIN {X 0,Y 601.428,Z 380.568,A -85,B 0,C 180,E1 -588.407,E2 -588.407} C_VEL
LIN {X 0,Y 601.433,Z 380.571,A -85,B 0,C 180,E1 -591.529,E2 -591.529} C_VEL
LIN {X 0,Y 601.379,Z 380.572,A -85,B 0,C 180,E1 -594.245,E2 -594.245} C_VEL
LIN {X 0,Y 601.395,Z 381.196,A -85,B 0,C 180,E1 -595.067,E2 -595.067} C_VEL
LIN {X 0,Y 601.434,Z 385.309,A -85,B 0,C 180,E1 -597.484,E2 -597.484} C_VEL
LIN {X 0,Y 601.377,Z 390.744,A -85,B 0,C 180,E1 -600.605,E2 -600.605} C_VEL
LIN {X 0,Y 601.389,Z 394.891,A -85,B 0,C 180,E1 -602.886,E2 -602.886} C_VEL
LIN {X 0,Y 601.377,Z 400.165,A -85,B 0,C 180,E1 -605.721,E2 -605.721} C_VEL
LIN {X 0,Y 601.355,Z 404.567,A -85,B 0,C 180,E1 -608.039,E2 -608.039} C_VEL
LIN {X 0,Y 601.353,Z 410.096,A -85,B 0,C 180,E1 -610.899,E2 -610.899} C_VEL
LIN {X 0,Y 601.353,Z 415.626,A -85,B 0,C 180,E1 -613.711,E2 -613.711} C_VEL
LIN {X 0,Y 601.331,Z 421.156,A -85,B 0,C 180,E1 -616.482,E2 -616.482} C_VEL
LIN {X 0,Y 601.353,Z 424.526,A -85,B 0,C 180,E1 -618.156,E2 -618.156} C_VEL
LIN {X 0,Y 601.607,Z 429.392,A -85,B 0,C 180,E1 -618.268,E2 -618.268} C_VEL
LIN {X 0,Y 601.557,Z 441.683,A -85,B 0,C 180,E1 -618.583,E2 -618.583} C_VEL
LIN {X 0,Y 601.545,Z 454.846,A -85,B 0,C 180,E1 -619.073,E2 -619.073} C_VEL
LIN {X 0,Y 601.481,Z 466.513,A -85,B 0,C 180,E1 -619.651,E2 -619.651} C_VEL
LIN {X 0,Y 601.47,Z 477.311,A -85,B 0,C 180,E1 -620.33,E2 -620.33} C_VEL
LIN {X 0,Y 601.435,Z 487.084,A -85,B 0,C 180,E1 -621.093,E2 -621.093} C_VEL
LIN {X 0,Y 601.407,Z 495.981,A -85,B 0,C 180,E1 -621.939,E2 -621.939} C_VEL
LIN {X 0,Y 601.407,Z 504.667,A -85,B 0,C 180,E1 -622.952,E2 -622.952} C_VEL
LIN {X 0,Y 601.361,Z 511.597,A -85,B 0,C 180,E1 -623.962,E2 -623.962} C_VEL
LIN {X 0,Y 601.344,Z 517.149,A -85,B 0,C 180,E1 -624.971,E2 -624.971} C_VEL
LIN {X 0,Y 601.347,Z 521.511,A -85,B 0,C 180,E1 -625.979,E2 -625.979} C_VEL
LIN {X 0,Y 601.344,Z 523.815,A -85,B 0,C 180,E1 -626.65,E2 -626.65} C_VEL
LIN {X 0,Y 601.324,Z 525.693,A -85,B 0,C 180,E1 -627.32,E2 -627.32} C_VEL
LIN {X 0,Y 601.343,Z 527.127,A -85,B 0,C 180,E1 -627.991,E2 -627.991} C_VEL
LIN {X 0,Y 601.339,Z 528.753,A -85,B 0,C 180,E1 -629.33,E2 -629.33} C_VEL
LIN {X 0,Y 601.336,Z 528.996,A -85,B 0,C 180,E1 -630,E2 -630} C_VEL
LIN {X 0,Y 601.339,Z 528.815,A -85,B 0,C 180,E1 -630.67,E2 -630.67} C_VEL
LIN {X 0,Y 601.343,Z 527.275,A -85,B 0,C 180,E1 -632.009,E2 -632.009} C_VEL
LIN {X 0,Y 601.326,Z 525.916,A -85,B 0,C 180,E1 -632.68,E2 -632.68} C_VEL
LIN {X 0,Y 601.368,Z 523.04,A -85,B 0,C 180,E1 -633.685,E2 -633.685} C_VEL
LIN {X 0,Y 601.337,Z 519.14,A -85,B 0,C 180,E1 -634.693,E2 -634.693} C_VEL
LIN {X 0,Y 601.373,Z 514.109,A -85,B 0,C 180,E1 -635.701,E2 -635.701} C_VEL
LIN {X 0,Y 601.382,Z 507.791,A -85,B 0,C 180,E1 -636.711,E2 -636.711} C_VEL
LIN {X 0,Y 601.396,Z 499.873,A -85,B 0,C 180,E1 -637.723,E2 -637.723} C_VEL
LIN {X 0,Y 601.437,Z 490.029,A -85,B 0,C 180,E1 -638.738,E2 -638.738} C_VEL
LIN {X 0,Y 601.451,Z 479.706,A -85,B 0,C 180,E1 -639.585,E2 -639.585} C_VEL
LIN {X 0,Y 601.481,Z 468.088,A -85,B 0,C 180,E1 -640.349,E2 -640.349} C_VEL
LIN {X 0,Y 601.523,Z 456.209,A -85,B 0,C 180,E1 -640.958,E2 -640.958} C_VEL
LIN {X 0,Y 601.543,Z 443.243,A -85,B 0,C 180,E1 -641.456,E2 -641.456} C_VEL
LIN {X 0,Y 601.615,Z 430.617,A -85,B 0,C 180,E1 -641.796,E2 -641.796} C_VEL
LIN {X 0,Y 601.348,Z 424.534,A -85,B 0,C 180,E1 -641.93,E2 -641.93} C_VEL
LIN {X 0,Y 601.341,Z 418.57,A -85,B 0,C 180,E1 -644.899,E2 -644.899} C_VEL
LIN {X 0,Y 601.34,Z 413.038,A -85,B 0,C 180,E1 -647.69,E2 -647.69} C_VEL
LIN {X 0,Y 601.344,Z 407.505,A -85,B 0,C 180,E1 -650.525,E2 -650.525} C_VEL
LIN {X 0,Y 601.368,Z 401.972,A -85,B 0,C 180,E1 -653.413,E2 -653.413} C_VEL
LIN {X 0,Y 601.36,Z 396.439,A -85,B 0,C 180,E1 -656.366,E2 -656.366} C_VEL
LIN {X 0,Y 601.369,Z 392.024,A -85,B 0,C 180,E1 -658.776,E2 -658.776} C_VEL
LIN {X 0,Y 601.382,Z 387.28,A -85,B 0,C 180,E1 -661.448,E2 -661.448} C_VEL
LIN {X 0,Y 601.426,Z 382.724,A -85,B 0,C 180,E1 -664.119,E2 -664.119} C_VEL
LIN {X 0,Y 601.38,Z 381.057,A -85,B 0,C 180,E1 -665.109,E2 -665.109} C_VEL
LIN {X 0,Y 601.38,Z 380.573,A -85,B 0,C 180,E1 -665.755,E2 -665.755} C_VEL
LIN {X 0,Y 601.433,Z 380.569,A -85,B 0,C 180,E1 -668.471,E2 -668.471} C_VEL
LIN {X 0,Y 601.428,Z 380.567,A -85,B 0,C 180,E1 -671.593,E2 -671.593} C_VEL
LIN {X 0,Y 601.429,Z 380.565,A -85,B 0,C 180,E1 -674.535,E2 -674.535} C_VEL
LIN {X 0,Y 601.41,Z 380.573,A -85,B 0,C 180,E1 -677.41,E2 -677.41} C_VEL
LIN {X 0,Y 601.444,Z 380.568,A -85,B 0,C 180,E1 -680.464,E2 -680.464} C_VEL
LIN {X 0,Y 601.406,Z 380.568,A -85,B 0,C 180,E1 -683.417,E2 -683.417} C_VEL
LIN {X 0,Y 601.436,Z 380.568,A -85,B 0,C 180,E1 -686.064,E2 -686.064} C_VEL
LIN {X 0,Y 601.423,Z 380.566,A -85,B 0,C 180,E1 -688.545,E2 -688.545} C_VEL
LIN {X 0,Y 601.428,Z 380.567,A -85,B 0,C 180,E1 -691.373,E2 -691.373} C_VEL
LIN {X 0,Y 601.404,Z 380.568,A -85,B 0,C 180,E1 -693.636,E2 -693.636} C_VEL
LIN {X 0,Y 601.462,Z 380.566,A -85,B 0,C 180,E1 -695.86,E2 -695.86} C_VEL
LIN {X 0,Y 601.408,Z 380.568,A -85,B 0,C 180,E1 -698.761,E2 -698.761} C_VEL
LIN {X 0,Y 601.419,Z 380.569,A -85,B 0,C 180,E1 -701.608,E2 -701.608} C_VEL
LIN {X 0,Y 601.416,Z 380.571,A -85,B 0,C 180,E1 -704.409,E2 -704.409} C_VEL
LIN {X 0,Y 601.422,Z 380.566,A -85,B 0,C 180,E1 -707.172,E2 -707.172} C_VEL
LIN {X 0,Y 601.431,Z 380.571,A -85,B 0,C 180,E1 -709.905,E2 -709.905} C_VEL
LIN {X 0,Y 601.444,Z 380.564,A -85,B 0,C 180,E1 -712.615,E2 -712.615} C_VEL
LIN {X 0,Y 601.424,Z 380.568,A -85,B 0,C 180,E1 -715.308,E2 -715.308} C_VEL
LIN {X 0,Y 601.419,Z 380.569,A -85,B 0,C 180,E1 -717.991,E2 -717.991} C_VEL
LIN {X 0,Y 601.45,Z 380.563,A -85,B 0,C 180,E1 -720.669,E2 -720.669} C_VEL
LIN {X 0,Y 601.429,Z 380.571,A -85,B 0,C 180,E1 -723.35,E2 -723.35} C_VEL
LIN {X 0,Y 601.408,Z 380.568,A -85,B 0,C 180,E1 -726.037,E2 -726.037} C_VEL
LIN {X 0,Y 601.443,Z 380.569,A -85,B 0,C 180,E1 -728.738,E2 -728.738} C_VEL
LIN {X 0,Y 601.437,Z 380.565,A -85,B 0,C 180,E1 -731.458,E2 -731.458} C_VEL
LIN {X 0,Y 601.423,Z 380.567,A -85,B 0,C 180,E1 -734.205,E2 -734.205} C_VEL
LIN {X 0,Y 601.425,Z 380.571,A -85,B 0,C 180,E1 -736.986,E2 -736.986} C_VEL
LIN {X 0,Y 601.41,Z 380.568,A -85,B 0,C 180,E1 -739.809,E2 -739.809} C_VEL
LIN {X 0,Y 601.415,Z 380.569,A -85,B 0,C 180,E1 -742.683,E2 -742.683} C_VEL
LIN {X 0,Y 601.404,Z 380.568,A -85,B 0,C 180,E1 -744.879,E2 -744.879} C_VEL
LIN {X 0,Y 601.425,Z 380.572,A -85,B 0,C 180,E1 -747.364,E2 -747.364} C_VEL
LIN {X 0,Y 601.432,Z 380.565,A -85,B 0,C 180,E1 -750.164,E2 -750.164} C_VEL
LIN {X 0,Y 601.424,Z 380.572,A -85,B 0,C 180,E1 -752.715,E2 -752.715} C_VEL
LIN {X 0,Y 601.4,Z 380.569,A -85,B 0,C 180,E1 -755.112,E2 -755.112} C_VEL
LIN {X 0,Y 601.436,Z 380.568,A -85,B 0,C 180,E1 -757.419,E2 -757.419} C_VEL
LIN {X 0,Y 601.415,Z 380.568,A -85,B 0,C 180,E1 -759.995,E2 -759.995} C_VEL
LIN {X 0,Y 601.411,Z 380.572,A -85,B 0,C 180,E1 -762.671,E2 -762.671} C_VEL
LIN {X 0,Y 601.43,Z 380.565,A -85,B 0,C 180,E1 -765.482,E2 -765.482} C_VEL
LIN {X 0,Y 601.428,Z 380.568,A -85,B 0,C 180,E1 -768.407,E2 -768.407} C_VEL
LIN {X 0,Y 601.432,Z 380.572,A -85,B 0,C 180,E1 -771.529,E2 -771.529} C_VEL
LIN {X 0,Y 601.438,Z 380.655,A -85,B 0,C 180,E1 -774.335,E2 -774.335} C_VEL
LIN {X 0,Y 601.526,Z 387.061,A -85,B 0,C 180,E1 -776.692,E2 -776.692} C_VEL
LIN {X 0,Y 601.487,Z 394.955,A -85,B 0,C 180,E1 -779.451,E2 -779.451} C_VEL
LIN {X 0,Y 601.453,Z 402.751,A -85,B 0,C 180,E1 -782.134,E2 -782.134} C_VEL
LIN {X 0,Y 601.425,Z 411.656,A -85,B 0,C 180,E1 -785.122,E2 -785.122} C_VEL
LIN {X 0,Y 601.42,Z 418.571,A -85,B 0,C 180,E1 -787.394,E2 -787.394} C_VEL
LIN {X 0,Y 601.41,Z 427.239,A -85,B 0,C 180,E1 -790.191,E2 -790.191} C_VEL
LIN {X 0,Y 601.372,Z 436.143,A -85,B 0,C 180,E1 -793.012,E2 -793.012} C_VEL
LIN {X 0,Y 601.362,Z 445.048,A -85,B 0,C 180,E1 -795.793,E2 -795.793} C_VEL
LIN {X 0,Y 601.38,Z 452.491,A -85,B 0,C 180,E1 -798.092,E2 -798.092} C_VEL
LIN {X 0,Y 601.599,Z 465.929,A -85,B 0,C 180,E1 -798.374,E2 -798.374} C_VEL
LIN {X 0,Y 601.55,Z 478.117,A -85,B 0,C 180,E1 -798.757,E2 -798.757} C_VEL
LIN {X 0,Y 601.513,Z 490.921,A -85,B 0,C 180,E1 -799.311,E2 -799.311} C_VEL
LIN {X 0,Y 601.477,Z 501.578,A -85,B 0,C 180,E1 -799.906,E2 -799.906} C_VEL
LIN {X 0,Y 601.449,Z 512.474,A -85,B 0,C 180,E1 -800.669,E2 -800.669} C_VEL
LIN {X 0,Y 601.429,Z 523.111,A -85,B 0,C 180,E1 -801.601,E2 -801.601} C_VEL
LIN {X 0,Y 601.418,Z 530.96,A -85,B 0,C 180,E1 -802.446,E2 -802.446} C_VEL
LIN {X 0,Y 601.37,Z 538.224,A -85,B 0,C 180,E1 -803.398,E2 -803.398} C_VEL
LIN {X 0,Y 601.372,Z 543.866,A -85,B 0,C 180,E1 -804.299,E2 -804.299} C_VEL
LIN {X 0,Y 601.336,Z 548.95,A -85,B 0,C 180,E1 -805.307,E2 -805.307} C_VEL
LIN {X 0,Y 601.367,Z 552.896,A -85,B 0,C 180,E1 -806.315,E2 -806.315} C_VEL
LIN {X 0,Y 601.325,Z 555.809,A -85,B 0,C 180,E1 -807.32,E2 -807.32} C_VEL
LIN {X 0,Y 601.343,Z 557.201,A -85,B 0,C 180,E1 -807.991,E2 -807.991} C_VEL
LIN {X 0,Y 601.339,Z 558.784,A -85,B 0,C 180,E1 -809.33,E2 -809.33} C_VEL
LIN {X 0,Y 601.335,Z 559,A -85,B 0,C 180,E1 -810,E2 -810} C_VEL
LIN {X 0,Y 601.348,Z 558.184,A -85,B 0,C 180,E1 -811.339,E2 -811.339} C_VEL
LIN {X 0,Y 601.343,Z 557.202,A -85,B 0,C 180,E1 -812.009,E2 -812.009} C_VEL
LIN {X 0,Y 601.325,Z 555.809,A -85,B 0,C 180,E1 -812.679,E2 -812.679} C_VEL
LIN {X 0,Y 601.367,Z 552.896,A -85,B 0,C 180,E1 -813.685,E2 -813.685} C_VEL
LIN {X 0,Y 601.336,Z 548.95,A -85,B 0,C 180,E1 -814.693,E2 -814.693} C_VEL
LIN {X 0,Y 601.372,Z 542.877,A -85,B 0,C 180,E1 -815.869,E2 -815.869} C_VEL
LIN {X 0,Y 601.382,Z 536.236,A -85,B 0,C 180,E1 -816.88,E2 -816.88} C_VEL
LIN {X 0,Y 601.4,Z 527.99,A -85,B 0,C 180,E1 -817.892,E2 -817.892} C_VEL
LIN {X 0,Y 601.436,Z 519.537,A -85,B 0,C 180,E1 -818.738,E2 -818.738} C_VEL
LIN {X 0,Y 601.451,Z 509.092,A -85,B 0,C 180,E1 -819.585,E2 -819.585} C_VEL
LIN {X 0,Y 601.469,Z 498.758,A -85,B 0,C 180,E1 -820.264,E2 -820.264} C_VEL
LIN {X 0,Y 601.538,Z 486.594,A -85,B 0,C 180,E1 -820.896,E2 -820.896} C_VEL
LIN {X 0,Y 601.57,Z 474.218,A -85,B 0,C 180,E1 -821.378,E2 -821.378} C_VEL
LIN {X 0,Y 601.611,Z 461.439,A -85,B 0,C 180,E1 -821.732,E2 -821.732} C_VEL
LIN {X 0,Y 601.38,Z 452.492,A -85,B 0,C 180,E1 -821.908,E2 -821.908} C_VEL
LIN {X 0,Y 601.364,Z 443.935,A -85,B 0,C 180,E1 -824.552,E2 -824.552} C_VEL
LIN {X 0,Y 601.39,Z 435.031,A -85,B 0,C 180,E1 -827.337,E2 -827.337} C_VEL
LIN {X 0,Y 601.395,Z 426.126,A -85,B 0,C 180,E1 -830.166,E2 -830.166} C_VEL
LIN {X 0,Y 601.424,Z 417.222,A -85,B 0,C 180,E1 -833.046,E2 -833.046} C_VEL
LIN {X 0,Y 601.439,Z 409.43,A -85,B 0,C 180,E1 -835.617,E2 -835.617} C_VEL
LIN {X 0,Y 601.458,Z 401.639,A -85,B 0,C 180,E1 -838.245,E2 -838.245} C_VEL
LIN {X 0,Y 601.469,Z 393.839,A -85,B 0,C 180,E1 -840.939,E2 -840.939} C_VEL
LIN {X 0,Y 601.525,Z 387.062,A -85,B 0,C 180,E1 -843.307,E2 -843.307} C_VEL
LIN {X 0,Y 601.435,Z 380.569,A -85,B 0,C 180,E1 -845.708,E2 -845.708} C_VEL
LIN {X 0,Y 601.43,Z 380.572,A -85,B 0,C 180,E1 -848.47,E2 -848.47} C_VEL
LIN {X 0,Y 601.428,Z 380.567,A -85,B 0,C 180,E1 -851.593,E2 -851.593} C_VEL
LIN {X 0,Y 601.427,Z 380.565,A -85,B 0,C 180,E1 -854.535,E2 -854.535} C_VEL
LIN {X 0,Y 601.41,Z 380.571,A -85,B 0,C 180,E1 -857.41,E2 -857.41} C_VEL
LIN {X 0,Y 601.443,Z 380.569,A -85,B 0,C 180,E1 -860.464,E2 -860.464} C_VEL
LIN {X 0,Y 601.413,Z 380.568,A -85,B 0,C 180,E1 -863.418,E2 -863.418} C_VEL
LIN {X 0,Y 601.434,Z 380.568,A -85,B 0,C 180,E1 -866.064,E2 -866.064} C_VEL
LIN {X 0,Y 601.422,Z 380.567,A -85,B 0,C 180,E1 -868.545,E2 -868.545} C_VEL
LIN {X 0,Y 601.428,Z 380.566,A -85,B 0,C 180,E1 -871.373,E2 -871.373} C_VEL
LIN {X 0,Y 601.405,Z 380.568,A -85,B 0,C 180,E1 -873.636,E2 -873.636} C_VEL
LIN {X 0,Y 601.463,Z 380.567,A -85,B 0,C 180,E1 -875.86,E2 -875.86} C_VEL
LIN {X 0,Y 601.405,Z 380.568,A -85,B 0,C 180,E1 -878.761,E2 -878.761} C_VEL
LIN {X 0,Y 601.42,Z 380.568,A -85,B 0,C 180,E1 -881.608,E2 -881.608} C_VEL
LIN {X 0,Y 601.417,Z 380.572,A -85,B 0,C 180,E1 -884.409,E2 -884.409} C_VEL
LIN {X 0,Y 601.422,Z 380.566,A -85,B 0,C 180,E1 -887.172,E2 -887.172} C_VEL
LIN {X 0,Y 601.428,Z 380.57,A -85,B 0,C 180,E1 -889.905,E2 -889.905} C_VEL
LIN {X 0,Y 601.442,Z 380.565,A -85,B 0,C 180,E1 -892.615,E2 -892.615} C_VEL
LIN {X 0,Y 601.427,Z 380.567,A -85,B 0,C 180,E1 -895.308,E2 -895.308} C_VEL
LIN {X 0,Y 601.424,Z 380.569,A -85,B 0,C 180,E1 -897.991,E2 -897.991} C_VEL
LIN {X 0,Y 601.449,Z 380.563,A -85,B 0,C 180,E1 -900.67,E2 -900.67} C_VEL
LIN {X 0,Y 601.428,Z 380.572,A -85,B 0,C 180,E1 -903.35,E2 -903.35} C_VEL
LIN {X 0,Y 601.408,Z 380.568,A -85,B 0,C 180,E1 -906.037,E2 -906.037} C_VEL
LIN {X 0,Y 601.443,Z 380.569,A -85,B 0,C 180,E1 -908.738,E2 -908.738} C_VEL
LIN {X 0,Y 601.438,Z 380.565,A -85,B 0,C 180,E1 -911.458,E2 -911.458} C_VEL
LIN {X 0,Y 601.412,Z 380.57,A -85,B 0,C 180,E1 -912.376,E2 -912.376} C_VEL
LIN {X 0,Y 600.746,Z 380.651,A -85,B 0,C 180,E1 -912.935,E2 -912.935} C_VEL
LIN {X 0,Y 597.895,Z 381.011,A -85,B 0,C 180,E1 -913.843,E2 -913.843} C_VEL
LIN {X 0,Y 595.485,Z 381.31,A -85,B 0,C 180,E1 -914.573,E2 -914.573} C_VEL
LIN {X 0,Y 594.448,Z 381.438,A -85,B 0,C 180,E1 -915.137,E2 -915.137} C_VEL
LIN {X 0,Y 594.362,Z 381.447,A -85,B 0,C 180,E1 -915.327,E2 -915.327} C_VEL
LIN {X 0,Y 594.386,Z 381.45,A -85,B 0,C 180,E1 -917.194,E2 -917.194} C_VEL
LIN {X 0,Y 594.378,Z 381.445,A -85,B 0,C 180,E1 -920.054,E2 -920.054} C_VEL
LIN {X 0,Y 594.36,Z 381.446,A -85,B 0,C 180,E1 -922.968,E2 -922.968} C_VEL
LIN {X 0,Y 594.382,Z 381.444,A -85,B 0,C 180,E1 -925.193,E2 -925.193} C_VEL
LIN {X 0,Y 594.389,Z 381.449,A -85,B 0,C 180,E1 -927.527,E2 -927.527} C_VEL
LIN {X 0,Y 594.389,Z 381.443,A -85,B 0,C 180,E1 -930.328,E2 -930.328} C_VEL
LIN {X 0,Y 594.379,Z 381.446,A -85,B 0,C 180,E1 -932.95,E2 -932.95} C_VEL
LIN {X 0,Y 594.385,Z 381.444,A -85,B 0,C 180,E1 -935.407,E2 -935.407} C_VEL
LIN {X 0,Y 594.388,Z 381.447,A -85,B 0,C 180,E1 -937.941,E2 -937.941} C_VEL
LIN {X 0,Y 594.379,Z 381.446,A -85,B 0,C 180,E1 -940.822,E2 -940.822} C_VEL
LIN {X 0,Y 594.368,Z 381.447,A -85,B 0,C 180,E1 -943.3,E2 -943.3} C_VEL
LIN {X 0,Y 594.386,Z 381.449,A -85,B 0,C 180,E1 -946.159,E2 -946.159} C_VEL
LIN {X 0,Y 594.379,Z 381.445,A -85,B 0,C 180,E1 -949.178,E2 -949.178} C_VEL
LIN {X 0,Y 594.387,Z 381.443,A -85,B 0,C 180,E1 -952.059,E2 -952.059} C_VEL
LIN {X 0,Y 594.308,Z 381.458,A -85,B 0,C 180,E1 -954.683,E2 -954.683} C_VEL
LIN {X 0,Y 594.347,Z 385.449,A -85,B 0,C 180,E1 -957.094,E2 -957.094} C_VEL
LIN {X 0,Y 594.315,Z 389.896,A -85,B 0,C 180,E1 -959.684,E2 -959.684} C_VEL
LIN {X 0,Y 594.335,Z 394.892,A -85,B 0,C 180,E1 -962.537,E2 -962.537} C_VEL
LIN {X 0,Y 594.299,Z 399.039,A -85,B 0,C 180,E1 -964.803,E2 -964.803} C_VEL
LIN {X 0,Y 594.276,Z 404.568,A -85,B 0,C 180,E1 -967.763,E2 -967.763} C_VEL
LIN {X 0,Y 594.246,Z 408.715,A -85,B 0,C 180,E1 -969.942,E2 -969.942} C_VEL
LIN {X 0,Y 594.294,Z 414.245,A -85,B 0,C 180,E1 -972.804,E2 -972.804} C_VEL
LIN {X 0,Y 594.261,Z 420.282,A -85,B 0,C 180,E1 -975.877,E2 -975.877} C_VEL
LIN {X 0,Y 594.277,Z 424.527,A -85,B 0,C 180,E1 -978.013,E2 -978.013} C_VEL
LIN {X 0,Y 594.665,Z 429.42,A -85,B 0,C 180,E1 -978.129,E2 -978.129} C_VEL
LIN {X 0,Y 594.59,Z 441.783,A -85,B 0,C 180,E1 -978.45,E2 -978.45} C_VEL
LIN {X 0,Y 594.56,Z 454.86,A -85,B 0,C 180,E1 -978.943,E2 -978.943} C_VEL
LIN {X 0,Y 594.5,Z 466.525,A -85,B 0,C 180,E1 -979.528,E2 -979.528} C_VEL
LIN {X 0,Y 594.448,Z 477.317,A -85,B 0,C 180,E1 -980.215,E2 -980.215} C_VEL
LIN {X 0,Y 594.404,Z 487.091,A -85,B 0,C 180,E1 -980.987,E2 -980.987} C_VEL
LIN {X 0,Y 594.366,Z 495.986,A -85,B 0,C 180,E1 -981.843,E2 -981.843} C_VEL
LIN {X 0,Y 594.345,Z 504.672,A -85,B 0,C 180,E1 -982.868,E2 -982.868} C_VEL
LIN {X 0,Y 594.29,Z 511.6,A -85,B 0,C 180,E1 -983.89,E2 -983.89} C_VEL
LIN {X 0,Y 594.253,Z 517.152,A -85,B 0,C 180,E1 -984.911,E2 -984.911} C_VEL
LIN {X 0,Y 594.263,Z 521.513,A -85,B 0,C 180,E1 -985.931,E2 -985.931} C_VEL
LIN {X 0,Y 594.267,Z 523.817,A -85,B 0,C 180,E1 -986.61,E2 -986.61} C_VEL
LIN {X 0,Y 594.225,Z 525.695,A -85,B 0,C 180,E1 -987.288,E2 -987.288} C_VEL
LIN {X 0,Y 594.242,Z 527.127,A -85,B 0,C 180,E1 -987.967,E2 -987.967} C_VEL
LIN {X 0,Y 594.24,Z 528.753,A -85,B 0,C 180,E1 -989.322,E2 -989.322} C_VEL
LIN {X 0,Y 594.236,Z 528.996,A -85,B 0,C 180,E1 -990,E2 -990} C_VEL
LIN {X 0,Y 594.239,Z 528.815,A -85,B 0,C 180,E1 -990.678,E2 -990.678} C_VEL
LIN {X 0,Y 594.242,Z 527.275,A -85,B 0,C 180,E1 -992.033,E2 -992.033} C_VEL
LIN {X 0,Y 594.226,Z 525.915,A -85,B 0,C 180,E1 -992.712,E2 -992.712} C_VEL
LIN {X 0,Y 594.289,Z 523.038,A -85,B 0,C 180,E1 -993.729,E2 -993.729} C_VEL
LIN {X 0,Y 594.241,Z 519.138,A -85,B 0,C 180,E1 -994.749,E2 -994.749} C_VEL
LIN {X 0,Y 594.3,Z 514.106,A -85,B 0,C 180,E1 -995.769,E2 -995.769} C_VEL
LIN {X 0,Y 594.316,Z 507.787,A -85,B 0,C 180,E1 -996.791,E2 -996.791} C_VEL
LIN {X 0,Y 594.346,Z 499.869,A -85,B 0,C 180,E1 -997.816,E2 -997.816} C_VEL
LIN {X 0,Y 594.381,Z 490.023,A -85,B 0,C 180,E1 -998.842,E2 -998.842} C_VEL
LIN {X 0,Y 594.435,Z 479.701,A -85,B 0,C 180,E1 -999.699,E2 -999.699} C_VEL
LIN {X 0,Y 594.5,Z 468.077,A -85,B 0,C 180,E1 -1000.472,E2 -1000.472} C_VEL
LIN {X 0,Y 594.565,Z 456.229,A -85,B 0,C 180,E1 -1001.087,E2 -1001.087} C_VEL
LIN {X 0,Y 594.582,Z 444.508,A -85,B 0,C 180,E1 -1001.549,E2 -1001.549} C_VEL
LIN {X 0,Y 594.644,Z 431.509,A -85,B 0,C 180,E1 -1001.915,E2 -1001.915} C_VEL
LIN {X 0,Y 594.495,Z 426.172,A -85,B 0,C 180,E1 -1002.026,E2 -1002.026} C_VEL
LIN {X 0,Y 594.261,Z 424.533,A -85,B 0,C 180,E1 -1002.074,E2 -1002.074} C_VEL
LIN {X 0,Y 594.261,Z 418.569,A -85,B 0,C 180,E1 -1005.081,E2 -1005.081} C_VEL
LIN {X 0,Y 594.258,Z 414.42,A -85,B 0,C 180,E1 -1007.197,E2 -1007.197} C_VEL
LIN {X 0,Y 594.244,Z 408.887,A -85,B 0,C 180,E1 -1010.058,E2 -1010.058} C_VEL
LIN {X 0,Y 594.309,Z 403.821,A -85,B 0,C 180,E1 -1012.721,E2 -1012.721} C_VEL
LIN {X 0,Y 594.298,Z 399.205,A -85,B 0,C 180,E1 -1015.197,E2 -1015.197} C_VEL
LIN {X 0,Y 594.311,Z 393.671,A -85,B 0,C 180,E1 -1018.231,E2 -1018.231} C_VEL
LIN {X 0,Y 594.3,Z 389.585,A -85,B 0,C 180,E1 -1020.564,E2 -1020.564} C_VEL
LIN {X 0,Y 594.348,Z 385.53,A -85,B 0,C 180,E1 -1022.952,E2 -1022.952} C_VEL
LIN {X 0,Y 594.309,Z 381.457,A -85,B 0,C 180,E1 -1025.412,E2 -1025.412} C_VEL
LIN {X 0,Y 594.388,Z 381.442,A -85,B 0,C 180,E1 -1027.941,E2 -1027.941} C_VEL
LIN {X 0,Y 594.379,Z 381.445,A -85,B 0,C 180,E1 -1030.822,E2 -1030.822} C_VEL
LIN {X 0,Y 594.387,Z 381.45,A -85,B 0,C 180,E1 -1033.841,E2 -1033.841} C_VEL
LIN {X 0,Y 594.368,Z 381.446,A -85,B 0,C 180,E1 -1036.7,E2 -1036.7} C_VEL
LIN {X 0,Y 594.37,Z 381.446,A -85,B 0,C 180,E1 -1039.433,E2 -1039.433} C_VEL
LIN {X 0,Y 594.392,Z 381.449,A -85,B 0,C 180,E1 -1042.392,E2 -1042.392} C_VEL
LIN {X 0,Y 594.386,Z 381.445,A -85,B 0,C 180,E1 -1045.42,E2 -1045.42} C_VEL
LIN {X 0,Y 594.38,Z 381.443,A -85,B 0,C 180,E1 -1048.357,E2 -1048.357} C_VEL
LIN {X 0,Y 594.385,Z 381.449,A -85,B 0,C 180,E1 -1051.042,E2 -1051.042} C_VEL
LIN {X 0,Y 594.389,Z 381.445,A -85,B 0,C 180,E1 -1053.977,E2 -1053.977} C_VEL
LIN {X 0,Y 594.382,Z 381.447,A -85,B 0,C 180,E1 -1056.295,E2 -1056.295} C_VEL
LIN {X 0,Y 594.408,Z 381.444,A -85,B 0,C 180,E1 -1059.224,E2 -1059.224} C_VEL
LIN {X 0,Y 594.355,Z 381.447,A -85,B 0,C 180,E1 -1062.095,E2 -1062.095} C_VEL
LIN {X 0,Y 594.369,Z 381.447,A -85,B 0,C 180,E1 -1064.219,E2 -1064.219} C_VEL
LIN {X 0,Y 594.384,Z 381.451,A -85,B 0,C 180,E1 -1066.321,E2 -1066.321} C_VEL
LIN {X 0,Y 594.376,Z 381.444,A -85,B 0,C 180,E1 -1069.095,E2 -1069.095} C_VEL
LIN {X 0,Y 594.417,Z 381.441,A -85,B 0,C 180,E1 -1071.843,E2 -1071.843} C_VEL
LIN {X 0,Y 594.397,Z 381.444,A -85,B 0,C 180,E1 -1074.572,E2 -1074.572} C_VEL
LIN {X 0,Y 594.41,Z 381.44,A -85,B 0,C 180,E1 -1077.289,E2 -1077.289} C_VEL
LIN {X 0,Y 594.415,Z 381.446,A -85,B 0,C 180,E1 -1080,E2 -1080} C_VEL
LIN {X 0,Y 594.41,Z 381.439,A -85,B 0,C 180,E1 -1082.711,E2 -1082.711} C_VEL
LIN {X 0,Y 594.394,Z 381.446,A -85,B 0,C 180,E1 -1085.428,E2 -1085.428} C_VEL
LIN {X 0,Y 594.417,Z 381.441,A -85,B 0,C 180,E1 -1088.157,E2 -1088.157} C_VEL
LIN {X 0,Y 594.39,Z 381.442,A -85,B 0,C 180,E1 -1091.072,E2 -1091.072} C_VEL
LIN {X 0,Y 594.389,Z 381.449,A -85,B 0,C 180,E1 -1093.679,E2 -1093.679} C_VEL
LIN {X 0,Y 594.394,Z 381.443,A -85,B 0,C 180,E1 -1096.718,E2 -1096.718} C_VEL
LIN {X 0,Y 594.372,Z 381.446,A -85,B 0,C 180,E1 -1099.334,E2 -1099.334} C_VEL
LIN {X 0,Y 594.367,Z 381.445,A -85,B 0,C 180,E1 -1101.503,E2 -1101.503} C_VEL
LIN {X 0,Y 594.393,Z 381.444,A -85,B 0,C 180,E1 -1104.446,E2 -1104.446} C_VEL
LIN {X 0,Y 594.39,Z 381.442,A -85,B 0,C 180,E1 -1106.699,E2 -1106.699} C_VEL
LIN {X 0,Y 594.383,Z 381.448,A -85,B 0,C 180,E1 -1108.998,E2 -1108.998} C_VEL
LIN {X 0,Y 594.381,Z 381.443,A -85,B 0,C 180,E1 -1111.643,E2 -1111.643} C_VEL
LIN {X 0,Y 594.385,Z 381.446,A -85,B 0,C 180,E1 -1114.58,E2 -1114.58} C_VEL
LIN {X 0,Y 594.391,Z 381.448,A -85,B 0,C 180,E1 -1117.608,E2 -1117.608} C_VEL
LIN {X 0,Y 594.37,Z 381.445,A -85,B 0,C 180,E1 -1120.567,E2 -1120.567} C_VEL
LIN {X 0,Y 594.369,Z 381.446,A -85,B 0,C 180,E1 -1123.3,E2 -1123.3} C_VEL
LIN {X 0,Y 594.387,Z 381.449,A -85,B 0,C 180,E1 -1126.159,E2 -1126.159} C_VEL
LIN {X 0,Y 594.378,Z 381.445,A -85,B 0,C 180,E1 -1129.178,E2 -1129.178} C_VEL
LIN {X 0,Y 594.386,Z 381.444,A -85,B 0,C 180,E1 -1132.059,E2 -1132.059} C_VEL
LIN {X 0,Y 594.391,Z 381.503,A -85,B 0,C 180,E1 -1134.177,E2 -1134.177} C_VEL
LIN {X 0,Y 594.481,Z 385.917,A -85,B 0,C 180,E1 -1135.848,E2 -1135.848} C_VEL
LIN {X 0,Y 594.475,Z 392.873,A -85,B 0,C 180,E1 -1138.343,E2 -1138.343} C_VEL
LIN {X 0,Y 594.456,Z 400.595,A -85,B 0,C 180,E1 -1141.03,E2 -1141.03} C_VEL
LIN {X 0,Y 594.4,Z 407.204,A -85,B 0,C 180,E1 -1143.301,E2 -1143.301} C_VEL
LIN {X 0,Y 594.42,Z 415.009,A -85,B 0,C 180,E1 -1145.931,E2 -1145.931} C_VEL
LIN {X 0,Y 594.354,Z 424.608,A -85,B 0,C 180,E1 -1149.091,E2 -1149.091} C_VEL
LIN {X 0,Y 594.338,Z 432.804,A -85,B 0,C 180,E1 -1151.738,E2 -1151.738} C_VEL
LIN {X 0,Y 594.316,Z 441.709,A -85,B 0,C 180,E1 -1154.569,E2 -1154.569} C_VEL
LIN {X 0,Y 594.294,Z 451.726,A -85,B 0,C 180,E1 -1157.71,E2 -1157.71} C_VEL
LIN {X 0,Y 594.292,Z 452.491,A -85,B 0,C 180,E1 -1157.948,E2 -1157.948} C_VEL
LIN {X 0,Y 594.676,Z 457.224,A -85,B 0,C 180,E1 -1158.042,E2 -1158.042} C_VEL
LIN {X 0,Y 594.626,Z 470.493,A -85,B 0,C 180,E1 -1158.366,E2 -1158.366} C_VEL
LIN {X 0,Y 594.57,Z 482.17,A -85,B 0,C 180,E1 -1158.781,E2 -1158.781} C_VEL
LIN {X 0,Y 594.515,Z 494.207,A -85,B 0,C 180,E1 -1159.356,E2 -1159.356} C_VEL
LIN {X 0,Y 594.475,Z 505.475,A -85,B 0,C 180,E1 -1160.043,E2 -1160.043} C_VEL
LIN {X 0,Y 594.406,Z 515.646,A -85,B 0,C 180,E1 -1160.815,E2 -1160.815} C_VEL
LIN {X 0,Y 594.372,Z 524.786,A -85,B 0,C 180,E1 -1161.671,E2 -1161.671} C_VEL
LIN {X 0,Y 594.316,Z 533.69,A -85,B 0,C 180,E1 -1162.697,E2 -1162.697} C_VEL
LIN {X 0,Y 594.281,Z 540.169,A -85,B 0,C 180,E1 -1163.615,E2 -1163.615} C_VEL
LIN {X 0,Y 594.289,Z 545.68,A -85,B 0,C 180,E1 -1164.571,E2 -1164.571} C_VEL
LIN {X 0,Y 594.27,Z 550.371,A -85,B 0,C 180,E1 -1165.591,E2 -1165.591} C_VEL
LIN {X 0,Y 594.267,Z 553.956,A -85,B 0,C 180,E1 -1166.61,E2 -1166.61} C_VEL
LIN {X 0,Y 594.226,Z 555.809,A -85,B 0,C 180,E1 -1167.288,E2 -1167.288} C_VEL
LIN {X 0,Y 594.242,Z 557.201,A -85,B 0,C 180,E1 -1167.967,E2 -1167.967} C_VEL
LIN {X 0,Y 594.239,Z 558.784,A -85,B 0,C 180,E1 -1169.322,E2 -1169.322} C_VEL
LIN {X 0,Y 594.236,Z 559,A -85,B 0,C 180,E1 -1170,E2 -1170} C_VEL
LIN {X 0,Y 594.248,Z 558.185,A -85,B 0,C 180,E1 -1171.355,E2 -1171.355} C_VEL
LIN {X 0,Y 594.242,Z 557.202,A -85,B 0,C 180,E1 -1172.033,E2 -1172.033} C_VEL
LIN {X 0,Y 594.226,Z 555.81,A -85,B 0,C 180,E1 -1172.712,E2 -1172.712} C_VEL
LIN {X 0,Y 594.288,Z 552.896,A -85,B 0,C 180,E1 -1173.729,E2 -1173.729} C_VEL
LIN {X 0,Y 594.241,Z 548.95,A -85,B 0,C 180,E1 -1174.749,E2 -1174.749} C_VEL
LIN {X 0,Y 594.304,Z 542.878,A -85,B 0,C 180,E1 -1175.939,E2 -1175.939} C_VEL
LIN {X 0,Y 594.308,Z 536.236,A -85,B 0,C 180,E1 -1176.962,E2 -1176.962} C_VEL
LIN {X 0,Y 594.359,Z 527.99,A -85,B 0,C 180,E1 -1177.986,E2 -1177.986} C_VEL
LIN {X 0,Y 594.382,Z 519.537,A -85,B 0,C 180,E1 -1178.842,E2 -1178.842} C_VEL
LIN {X 0,Y 594.435,Z 509.094,A -85,B 0,C 180,E1 -1179.699,E2 -1179.699} C_VEL
LIN {X 0,Y 594.482,Z 498.759,A -85,B 0,C 180,E1 -1180.386,E2 -1180.386} C_VEL
LIN {X 0,Y 594.557,Z 487.73,A -85,B 0,C 180,E1 -1180.973,E2 -1180.973} C_VEL
LIN {X 0,Y 594.59,Z 475.713,A -85,B 0,C 180,E1 -1181.464,E2 -1181.464} C_VEL
LIN {X 0,Y 594.657,Z 462.352,A -85,B 0,C 180,E1 -1181.85,E2 -1181.85} C_VEL
LIN {X 0,Y 594.43,Z 453.615,A -85,B 0,C 180,E1 -1182.028,E2 -1182.028} C_VEL
LIN {X 0,Y 594.298,Z 452.422,A -85,B 0,C 180,E1 -1182.074,E2 -1182.074} C_VEL
LIN {X 0,Y 594.295,Z 442.822,A -85,B 0,C 180,E1 -1185.08,E2 -1185.08} C_VEL
LIN {X 0,Y 594.33,Z 433.918,A -85,B 0,C 180,E1 -1187.906,E2 -1187.906} C_VEL
LIN {X 0,Y 594.357,Z 425.013,A -85,B 0,C 180,E1 -1190.777,E2 -1190.777} C_VEL
LIN {X 0,Y 594.398,Z 416.109,A -85,B 0,C 180,E1 -1193.704,E2 -1193.704} C_VEL
LIN {X 0,Y 594.409,Z 409.182,A -85,B 0,C 180,E1 -1196.027,E2 -1196.027} C_VEL
LIN {X 0,Y 594.447,Z 401.674,A -85,B 0,C 180,E1 -1198.596,E2 -1198.596} C_VEL
LIN {X 0,Y 594.457,Z 393.764,A -85,B 0,C 180,E1 -1201.345,E2 -1201.345} C_VEL
LIN {X 0,Y 594.504,Z 386.997,A -85,B 0,C 180,E1 -1203.753,E2 -1203.753} C_VEL
LIN {X 0,Y 594.548,Z 382.598,A -85,B 0,C 180,E1 -1205.396,E2 -1205.396} C_VEL
LIN {X 0,Y 594.376,Z 381.449,A -85,B 0,C 180,E1 -1205.928,E2 -1205.928} C_VEL
LIN {X 0,Y 594.378,Z 381.449,A -85,B 0,C 180,E1 -1208.805,E2 -1208.805} C_VEL
LIN {X 0,Y 594.388,Z 381.448,A -85,B 0,C 180,E1 -1211.849,E2 -1211.849} C_VEL
LIN {X 0,Y 594.385,Z 381.444,A -85,B 0,C 180,E1 -1214.236,E2 -1214.236} C_VEL
LIN {X 0,Y 594.361,Z 381.454,A -85,B 0,C 180,E1 -1217.148,E2 -1217.148} C_VEL
LIN {X 0,Y 594.369,Z 381.445,A -85,B 0,C 180,E1 -1219.433,E2 -1219.433} C_VEL
LIN {X 0,Y 594.39,Z 381.449,A -85,B 0,C 180,E1 -1222.392,E2 -1222.392} C_VEL
LIN {X 0,Y 594.358,Z 381.447,A -85,B 0,C 180,E1 -1224.676,E2 -1224.676} C_VEL
LIN {X 0,Y 594.381,Z 381.446,A -85,B 0,C 180,E1 -1227.088,E2 -1227.088} C_VEL
LIN {X 0,Y 594.389,Z 381.443,A -85,B 0,C 180,E1 -1229.672,E2 -1229.672} C_VEL
LIN {X 0,Y 594.377,Z 381.451,A -85,B 0,C 180,E1 -1232.539,E2 -1232.539} C_VEL
LIN {X 0,Y 594.379,Z 381.445,A -85,B 0,C 180,E1 -1234.807,E2 -1234.807} C_VEL
LIN {X 0,Y 594.364,Z 381.447,A -85,B 0,C 180,E1 -1237.265,E2 -1237.265} C_VEL
LIN {X 0,Y 594.379,Z 381.445,A -85,B 0,C 180,E1 -1239.946,E2 -1239.946} C_VEL
LIN {X 0,Y 594.391,Z 381.449,A -85,B 0,C 180,E1 -1242.807,E2 -1242.807} C_VEL
LIN {X 0,Y 594.392,Z 381.443,A -85,B 0,C 180,E1 -1245.826,E2 -1245.826} C_VEL
LIN {X 0,Y 594.397,Z 381.444,A -85,B 0,C 180,E1 -1248.404,E2 -1248.404} C_VEL
LIN {X 0,Y 594.401,Z 381.444,A -85,B 0,C 180,E1 -1251.158,E2 -1251.158} C_VEL
LIN {X 0,Y 594.365,Z 381.445,A -85,B 0,C 180,E1 -1253.891,E2 -1253.891} C_VEL
LIN {X 0,Y 594.379,Z 381.451,A -85,B 0,C 180,E1 -1256.611,E2 -1256.611} C_VEL
LIN {X 0,Y 594.421,Z 381.438,A -85,B 0,C 180,E1 -1259.323,E2 -1259.323} C_VEL
LIN {X 0,Y 594.39,Z 381.445,A -85,B 0,C 180,E1 -1262.033,E2 -1262.033} C_VEL
LIN {X 0,Y 594.396,Z 381.444,A -85,B 0,C 180,E1 -1264.748,E2 -1264.748} C_VEL
LIN {X 0,Y 594.397,Z 381.442,A -85,B 0,C 180,E1 -1267.473,E2 -1267.473} C_VEL
LIN {X 0,Y 594.39,Z 381.449,A -85,B 0,C 180,E1 -1270.216,E2 -1270.216} C_VEL
LIN {X 0,Y 594.37,Z 381.444,A -85,B 0,C 180,E1 -1272.983,E2 -1272.983} C_VEL
LIN {X 0,Y 594.362,Z 381.447,A -85,B 0,C 180,E1 -1275.327,E2 -1275.327} C_VEL
LIN {X 0,Y 593.686,Z 381.533,A -85,B 0,C 180,E1 -1275.893,E2 -1275.893} C_VEL
LIN {X 0,Y 590.816,Z 381.89,A -85,B 0,C 180,E1 -1276.811,E2 -1276.811} C_VEL
LIN {X 0,Y 588.404,Z 382.19,A -85,B 0,C 180,E1 -1277.55,E2 -1277.55} C_VEL
LIN {X 0,Y 587.382,Z 382.316,A -85,B 0,C 180,E1 -1278.12,E2 -1278.12} C_VEL
LIN {X 0,Y 587.306,Z 382.326,A -85,B 0,C 180,E1 -1278.313,E2 -1278.313} C_VEL
LIN {X 0,Y 587.333,Z 382.323,A -85,B 0,C 180,E1 -1281.038,E2 -1281.038} C_VEL
LIN {X 0,Y 587.318,Z 382.323,A -85,B 0,C 180,E1 -1283.259,E2 -1283.259} C_VEL
LIN {X 0,Y 587.34,Z 382.325,A -85,B 0,C 180,E1 -1285.517,E2 -1285.517} C_VEL
LIN {X 0,Y 587.349,Z 382.322,A -85,B 0,C 180,E1 -1287.818,E2 -1287.818} C_VEL
LIN {X 0,Y 587.34,Z 382.323,A -85,B 0,C 180,E1 -1290.51,E2 -1290.51} C_VEL
LIN {X 0,Y 587.335,Z 382.321,A -85,B 0,C 180,E1 -1293.397,E2 -1293.397} C_VEL
LIN {X 0,Y 587.359,Z 382.324,A -85,B 0,C 180,E1 -1295.896,E2 -1295.896} C_VEL
LIN {X 0,Y 587.335,Z 382.321,A -85,B 0,C 180,E1 -1298.479,E2 -1298.479} C_VEL
LIN {X 0,Y 587.338,Z 382.328,A -85,B 0,C 180,E1 -1301.157,E2 -1301.157} C_VEL
LIN {X 0,Y 587.314,Z 382.325,A -85,B 0,C 180,E1 -1304.112,E2 -1304.112} C_VEL
LIN {X 0,Y 587.325,Z 382.323,A -85,B 0,C 180,E1 -1306.994,E2 -1306.994} C_VEL
LIN {X 0,Y 587.315,Z 382.33,A -85,B 0,C 180,E1 -1309.746,E2 -1309.746} C_VEL
LIN {X 0,Y 587.347,Z 382.319,A -85,B 0,C 180,E1 -1312.392,E2 -1312.392} C_VEL
LIN {X 0,Y 587.261,Z 382.333,A -85,B 0,C 180,E1 -1314.468,E2 -1314.468} C_VEL
LIN {X 0,Y 587.291,Z 382.699,A -85,B 0,C 180,E1 -1314.942,E2 -1314.942} C_VEL
LIN {X 0,Y 587.298,Z 386.815,A -85,B 0,C 180,E1 -1317.418,E2 -1317.418} C_VEL
LIN {X 0,Y 587.259,Z 390.885,A -85,B 0,C 180,E1 -1319.826,E2 -1319.826} C_VEL
LIN {X 0,Y 587.264,Z 395.19,A -85,B 0,C 180,E1 -1322.324,E2 -1322.324} C_VEL
LIN {X 0,Y 587.228,Z 400.422,A -85,B 0,C 180,E1 -1325.236,E2 -1325.236} C_VEL
LIN {X 0,Y 587.222,Z 404.569,A -85,B 0,C 180,E1 -1327.481,E2 -1327.481} C_VEL
LIN {X 0,Y 587.182,Z 408.716,A -85,B 0,C 180,E1 -1329.69,E2 -1329.69} C_VEL
LIN {X 0,Y 587.17,Z 412.863,A -85,B 0,C 180,E1 -1331.868,E2 -1331.868} C_VEL
LIN {X 0,Y 587.171,Z 417.011,A -85,B 0,C 180,E1 -1334.021,E2 -1334.021} C_VEL
LIN {X 0,Y 587.18,Z 421.158,A -85,B 0,C 180,E1 -1336.15,E2 -1336.15} C_VEL
LIN {X 0,Y 587.166,Z 424.528,A -85,B 0,C 180,E1 -1337.865,E2 -1337.865} C_VEL
LIN {X 0,Y 587.712,Z 429.447,A -85,B 0,C 180,E1 -1337.986,E2 -1337.986} C_VEL
LIN {X 0,Y 587.639,Z 441.894,A -85,B 0,C 180,E1 -1338.315,E2 -1338.315} C_VEL
LIN {X 0,Y 587.589,Z 454.874,A -85,B 0,C 180,E1 -1338.811,E2 -1338.811} C_VEL
LIN {X 0,Y 587.521,Z 466.537,A -85,B 0,C 180,E1 -1339.402,E2 -1339.402} C_VEL
LIN {X 0,Y 587.445,Z 477.323,A -85,B 0,C 180,E1 -1340.097,E2 -1340.097} C_VEL
LIN {X 0,Y 587.357,Z 487.098,A -85,B 0,C 180,E1 -1340.878,E2 -1340.878} C_VEL
LIN {X 0,Y 587.302,Z 495.991,A -85,B 0,C 180,E1 -1341.744,E2 -1341.744} C_VEL
LIN {X 0,Y 587.274,Z 504.676,A -85,B 0,C 180,E1 -1342.781,E2 -1342.781} C_VEL
LIN {X 0,Y 587.214,Z 511.604,A -85,B 0,C 180,E1 -1343.816,E2 -1343.816} C_VEL
LIN {X 0,Y 587.167,Z 517.154,A -85,B 0,C 180,E1 -1344.85,E2 -1344.85} C_VEL
LIN {X 0,Y 587.182,Z 521.516,A -85,B 0,C 180,E1 -1345.882,E2 -1345.882} C_VEL
LIN {X 0,Y 587.193,Z 523.819,A -85,B 0,C 180,E1 -1346.569,E2 -1346.569} C_VEL
LIN {X 0,Y 587.131,Z 525.696,A -85,B 0,C 180,E1 -1347.256,E2 -1347.256} C_VEL
LIN {X 0,Y 587.141,Z 527.128,A -85,B 0,C 180,E1 -1347.942,E2 -1347.942} C_VEL
LIN {X 0,Y 587.14,Z 528.754,A -85,B 0,C 180,E1 -1349.314,E2 -1349.314} C_VEL
LIN {X 0,Y 587.137,Z 528.996,A -85,B 0,C 180,E1 -1350,E2 -1350} C_VEL
LIN {X 0,Y 587.14,Z 528.815,A -85,B 0,C 180,E1 -1350.686,E2 -1350.686} C_VEL
LIN {X 0,Y 587.141,Z 527.274,A -85,B 0,C 180,E1 -1352.058,E2 -1352.058} C_VEL
LIN {X 0,Y 587.133,Z 525.913,A -85,B 0,C 180,E1 -1352.744,E2 -1352.744} C_VEL
LIN {X 0,Y 587.213,Z 523.036,A -85,B 0,C 180,E1 -1353.774,E2 -1353.774} C_VEL
LIN {X 0,Y 587.147,Z 519.136,A -85,B 0,C 180,E1 -1354.806,E2 -1354.806} C_VEL
LIN {X 0,Y 587.23,Z 514.104,A -85,B 0,C 180,E1 -1355.839,E2 -1355.839} C_VEL
LIN {X 0,Y 587.23,Z 507.783,A -85,B 0,C 180,E1 -1356.874,E2 -1356.874} C_VEL
LIN {X 0,Y 587.288,Z 499.864,A -85,B 0,C 180,E1 -1357.91,E2 -1357.91} C_VEL
LIN {X 0,Y 587.343,Z 490.017,A -85,B 0,C 180,E1 -1358.949,E2 -1358.949} C_VEL
LIN {X 0,Y 587.422,Z 479.695,A -85,B 0,C 180,E1 -1359.816,E2 -1359.816} C_VEL
LIN {X 0,Y 587.497,Z 469.487,A -85,B 0,C 180,E1 -1360.511,E2 -1360.511} C_VEL
LIN {X 0,Y 587.59,Z 457.125,A -85,B 0,C 180,E1 -1361.179,E2 -1361.179} C_VEL
LIN {X 0,Y 587.631,Z 444.441,A -85,B 0,C 180,E1 -1361.69,E2 -1361.69} C_VEL
LIN {X 0,Y 587.717,Z 431.485,A -85,B 0,C 180,E1 -1362.058,E2 -1362.058} C_VEL
LIN {X 0,Y 587.402,Z 426.142,A -85,B 0,C 180,E1 -1362.174,E2 -1362.174} C_VEL
LIN {X 0,Y 587.162,Z 424.532,A -85,B 0,C 180,E1 -1362.223,E2 -1362.223} C_VEL
LIN {X 0,Y 587.182,Z 419.951,A -85,B 0,C 180,E1 -1364.558,E2 -1364.558} C_VEL
LIN {X 0,Y 587.186,Z 414.419,A -85,B 0,C 180,E1 -1367.411,E2 -1367.411} C_VEL
LIN {X 0,Y 587.188,Z 410.269,A -85,B 0,C 180,E1 -1369.581,E2 -1369.581} C_VEL
LIN {X 0,Y 587.191,Z 406.12,A -85,B 0,C 180,E1 -1371.78,E2 -1371.78} C_VEL
LIN {X 0,Y 587.205,Z 400.985,A -85,B 0,C 180,E1 -1374.548,E2 -1374.548} C_VEL
LIN {X 0,Y 587.225,Z 396.437,A -85,B 0,C 180,E1 -1377.052,E2 -1377.052} C_VEL
LIN {X 0,Y 587.228,Z 392.38,A -85,B 0,C 180,E1 -1379.386,E2 -1379.386} C_VEL
LIN {X 0,Y 587.317,Z 388.234,A -85,B 0,C 180,E1 -1381.831,E2 -1381.831} C_VEL
LIN {X 0,Y 587.337,Z 384.011,A -85,B 0,C 180,E1 -1384.346,E2 -1384.346} C_VEL
LIN {X 0,Y 587.263,Z 382.333,A -85,B 0,C 180,E1 -1385.533,E2 -1385.533} C_VEL
LIN {X 0,Y 587.342,Z 382.32,A -85,B 0,C 180,E1 -1387.838,E2 -1387.838} C_VEL
LIN {X 0,Y 587.314,Z 382.329,A -85,B 0,C 180,E1 -1390.255,E2 -1390.255} C_VEL
LIN {X 0,Y 587.325,Z 382.322,A -85,B 0,C 180,E1 -1393.006,E2 -1393.006} C_VEL
LIN {X 0,Y 587.315,Z 382.326,A -85,B 0,C 180,E1 -1395.888,E2 -1395.888} C_VEL
LIN {X 0,Y 587.339,Z 382.328,A -85,B 0,C 180,E1 -1398.925,E2 -1398.925} C_VEL
LIN {X 0,Y 587.336,Z 382.321,A -85,B 0,C 180,E1 -1401.521,E2 -1401.521} C_VEL
LIN {X 0,Y 587.296,Z 382.333,A -85,B 0,C 180,E1 -1404.1,E2 -1404.1} C_VEL
LIN {X 0,Y 587.336,Z 382.321,A -85,B 0,C 180,E1 -1406.603,E2 -1406.603} C_VEL
LIN {X 0,Y 587.34,Z 382.324,A -85,B 0,C 180,E1 -1409.49,E2 -1409.49} C_VEL
LIN {X 0,Y 587.355,Z 382.322,A -85,B 0,C 180,E1 -1412.307,E2 -1412.307} C_VEL
LIN {X 0,Y 587.339,Z 382.326,A -85,B 0,C 180,E1 -1414.483,E2 -1414.483} C_VEL
LIN {X 0,Y 587.343,Z 382.323,A -85,B 0,C 180,E1 -1417.486,E2 -1417.486} C_VEL
LIN {X 0,Y 587.347,Z 382.32,A -85,B 0,C 180,E1 -1420.425,E2 -1420.425} C_VEL
LIN {X 0,Y 587.351,Z 382.321,A -85,B 0,C 180,E1 -1423.311,E2 -1423.311} C_VEL
LIN {X 0,Y 587.362,Z 382.323,A -85,B 0,C 180,E1 -1426.154,E2 -1426.154} C_VEL
LIN {X 0,Y 587.342,Z 382.32,A -85,B 0,C 180,E1 -1428.962,E2 -1428.962} C_VEL
LIN {X 0,Y 587.371,Z 382.32,A -85,B 0,C 180,E1 -1431.745,E2 -1431.745} C_VEL
LIN {X 0,Y 587.361,Z 382.32,A -85,B 0,C 180,E1 -1434.507,E2 -1434.507} C_VEL
LIN {X 0,Y 587.376,Z 382.316,A -85,B 0,C 180,E1 -1437.257,E2 -1437.257} C_VEL
LIN {X 0,Y 587.385,Z 382.322,A -85,B 0,C 180,E1 -1440,E2 -1440} C_VEL
LIN {X 0,Y 587.377,Z 382.316,A -85,B 0,C 180,E1 -1442.743,E2 -1442.743} C_VEL
LIN {X 0,Y 587.358,Z 382.321,A -85,B 0,C 180,E1 -1445.493,E2 -1445.493} C_VEL
LIN {X 0,Y 587.372,Z 382.319,A -85,B 0,C 180,E1 -1448.255,E2 -1448.255} C_VEL
LIN {X 0,Y 587.352,Z 382.319,A -85,B 0,C 180,E1 -1451.134,E2 -1451.134} C_VEL
LIN {X 0,Y 587.37,Z 382.318,A -85,B 0,C 180,E1 -1454.261,E2 -1454.261} C_VEL
LIN {X 0,Y 587.35,Z 382.323,A -85,B 0,C 180,E1 -1457.406,E2 -1457.406} C_VEL
LIN {X 0,Y 587.334,Z 382.325,A -85,B 0,C 180,E1 -1460.305,E2 -1460.305} C_VEL
LIN {X 0,Y 587.318,Z 382.323,A -85,B 0,C 180,E1 -1463.259,E2 -1463.259} C_VEL
LIN {X 0,Y 587.338,Z 382.325,A -85,B 0,C 180,E1 -1465.517,E2 -1465.517} C_VEL
LIN {X 0,Y 587.35,Z 382.321,A -85,B 0,C 180,E1 -1467.818,E2 -1467.818} C_VEL
LIN {X 0,Y 587.341,Z 382.323,A -85,B 0,C 180,E1 -1470.51,E2 -1470.51} C_VEL
LIN {X 0,Y 587.336,Z 382.321,A -85,B 0,C 180,E1 -1473.397,E2 -1473.397} C_VEL
LIN {X 0,Y 587.302,Z 382.332,A -85,B 0,C 180,E1 -1475.899,E2 -1475.899} C_VEL
LIN {X 0,Y 587.334,Z 382.321,A -85,B 0,C 180,E1 -1478.479,E2 -1478.479} C_VEL
LIN {X 0,Y 587.339,Z 382.328,A -85,B 0,C 180,E1 -1481.157,E2 -1481.157} C_VEL
LIN {X 0,Y 587.33,Z 382.323,A -85,B 0,C 180,E1 -1484.113,E2 -1484.113} C_VEL
LIN {X 0,Y 587.325,Z 382.323,A -85,B 0,C 180,E1 -1486.994,E2 -1486.994} C_VEL
LIN {X 0,Y 587.314,Z 382.331,A -85,B 0,C 180,E1 -1489.745,E2 -1489.745} C_VEL
LIN {X 0,Y 587.347,Z 382.321,A -85,B 0,C 180,E1 -1492.392,E2 -1492.392} C_VEL
LIN {X 0,Y 587.361,Z 382.424,A -85,B 0,C 180,E1 -1494.052,E2 -1494.052} C_VEL
LIN {X 0,Y 587.477,Z 386.947,A -85,B 0,C 180,E1 -1495.787,E2 -1495.787} C_VEL
LIN {X 0,Y 587.475,Z 393.681,A -85,B 0,C 180,E1 -1498.239,E2 -1498.239} C_VEL
LIN {X 0,Y 587.456,Z 401.096,A -85,B 0,C 180,E1 -1500.849,E2 -1500.849} C_VEL
LIN {X 0,Y 587.374,Z 409.703,A -85,B 0,C 180,E1 -1503.817,E2 -1503.817} C_VEL
LIN {X 0,Y 587.346,Z 417.221,A -85,B 0,C 180,E1 -1506.368,E2 -1506.368} C_VEL
LIN {X 0,Y 587.302,Z 426.141,A -85,B 0,C 180,E1 -1509.333,E2 -1509.333} C_VEL
LIN {X 0,Y 587.282,Z 435.03,A -85,B 0,C 180,E1 -1512.232,E2 -1512.232} C_VEL
LIN {X 0,Y 587.223,Z 443.935,A -85,B 0,C 180,E1 -1515.089,E2 -1515.089} C_VEL
LIN {X 0,Y 587.197,Z 452.491,A -85,B 0,C 180,E1 -1517.8,E2 -1517.8} C_VEL
LIN {X 0,Y 587.757,Z 457.224,A -85,B 0,C 180,E1 -1517.899,E2 -1517.899} C_VEL
LIN {X 0,Y 587.696,Z 470.493,A -85,B 0,C 180,E1 -1518.226,E2 -1518.226} C_VEL
LIN {X 0,Y 587.591,Z 483.174,A -85,B 0,C 180,E1 -1518.69,E2 -1518.69} C_VEL
LIN {X 0,Y 587.533,Z 494.209,A -85,B 0,C 180,E1 -1519.228,E2 -1519.228} C_VEL
LIN {X 0,Y 587.463,Z 505.477,A -85,B 0,C 180,E1 -1519.923,E2 -1519.923} C_VEL
LIN {X 0,Y 587.384,Z 515.646,A -85,B 0,C 180,E1 -1520.704,E2 -1520.704} C_VEL
LIN {X 0,Y 587.34,Z 524.786,A -85,B 0,C 180,E1 -1521.571,E2 -1521.571} C_VEL
LIN {X 0,Y 587.259,Z 533.69,A -85,B 0,C 180,E1 -1522.608,E2 -1522.608} C_VEL
LIN {X 0,Y 587.195,Z 540.745,A -85,B 0,C 180,E1 -1523.627,E2 -1523.627} C_VEL
LIN {X 0,Y 587.211,Z 545.68,A -85,B 0,C 180,E1 -1524.506,E2 -1524.506} C_VEL
LIN {X 0,Y 587.188,Z 550.371,A -85,B 0,C 180,E1 -1525.538,E2 -1525.538} C_VEL
LIN {X 0,Y 587.193,Z 553.956,A -85,B 0,C 180,E1 -1526.569,E2 -1526.569} C_VEL
LIN {X 0,Y 587.132,Z 555.808,A -85,B 0,C 180,E1 -1527.256,E2 -1527.256} C_VEL
LIN {X 0,Y 587.141,Z 557.2,A -85,B 0,C 180,E1 -1527.942,E2 -1527.942} C_VEL
LIN {X 0,Y 587.14,Z 558.784,A -85,B 0,C 180,E1 -1529.314,E2 -1529.314} C_VEL
LIN {X 0,Y 587.137,Z 559,A -85,B 0,C 180,E1 -1530,E2 -1530} C_VEL
LIN {X 0,Y 587.147,Z 558.185,A -85,B 0,C 180,E1 -1531.372,E2 -1531.372} C_VEL
LIN {X 0,Y 587.141,Z 557.201,A -85,B 0,C 180,E1 -1532.058,E2 -1532.058} C_VEL
LIN {X 0,Y 587.132,Z 555.81,A -85,B 0,C 180,E1 -1532.744,E2 -1532.744} C_VEL
LIN {X 0,Y 587.212,Z 552.896,A -85,B 0,C 180,E1 -1533.774,E2 -1533.774} C_VEL
LIN {X 0,Y 587.147,Z 548.95,A -85,B 0,C 180,E1 -1534.806,E2 -1534.806} C_VEL
LIN {X 0,Y 587.217,Z 542.878,A -85,B 0,C 180,E1 -1536.011,E2 -1536.011} C_VEL
LIN {X 0,Y 587.245,Z 536.237,A -85,B 0,C 180,E1 -1537.046,E2 -1537.046} C_VEL
LIN {X 0,Y 587.299,Z 527.99,A -85,B 0,C 180,E1 -1538.083,E2 -1538.083} C_VEL
LIN {X 0,Y 587.343,Z 519.538,A -85,B 0,C 180,E1 -1538.949,E2 -1538.949} C_VEL
LIN {X 0,Y 587.422,Z 509.095,A -85,B 0,C 180,E1 -1539.816,E2 -1539.816} C_VEL
LIN {X 0,Y 587.486,Z 498.759,A -85,B 0,C 180,E1 -1540.511,E2 -1540.511} C_VEL
LIN {X 0,Y 587.561,Z 486.816,A -85,B 0,C 180,E1 -1541.149,E2 -1541.149} C_VEL
LIN {X 0,Y 587.632,Z 474.599,A -85,B 0,C 180,E1 -1541.639,E2 -1541.639} C_VEL
LIN {X 0,Y 587.709,Z 461.437,A -85,B 0,C 180,E1 -1542.014,E2 -1542.014} C_VEL
LIN {X 0,Y 587.546,Z 454.651,A -85,B 0,C 180,E1 -1542.154,E2 -1542.154} C_VEL
LIN {X 0,Y 587.197,Z 452.492,A -85,B 0,C 180,E1 -1542.2,E2 -1542.2} C_VEL
LIN {X 0,Y 587.223,Z 443.935,A -85,B 0,C 180,E1 -1544.911,E2 -1544.911} C_VEL
LIN {X 0,Y 587.282,Z 435.031,A -85,B 0,C 180,E1 -1547.768,E2 -1547.768} C_VEL
LIN {X 0,Y 587.302,Z 426.141,A -85,B 0,C 180,E1 -1550.667,E2 -1550.667} C_VEL
LIN {X 0,Y 587.345,Z 417.222,A -85,B 0,C 180,E1 -1553.631,E2 -1553.631} C_VEL
LIN {X 0,Y 587.373,Z 409.43,A -85,B 0,C 180,E1 -1556.277,E2 -1556.277} C_VEL
LIN {X 0,Y 587.469,Z 400.459,A -85,B 0,C 180,E1 -1559.373,E2 -1559.373} C_VEL
LIN {X 0,Y 587.484,Z 392.52,A -85,B 0,C 180,E1 -1562.175,E2 -1562.175} C_VEL
LIN {X 0,Y 587.503,Z 386.527,A -85,B 0,C 180,E1 -1564.369,E2 -1564.369} C_VEL
LIN {X 0,Y 587.336,Z 382.327,A -85,B 0,C 180,E1 -1566.003,E2 -1566.003} C_VEL
LIN {X 0,Y 587.329,Z 382.329,A -85,B 0,C 180,E1 -1568.479,E2 -1568.479} C_VEL
LIN {X 0,Y 587.339,Z 382.321,A -85,B 0,C 180,E1 -1571.157,E2 -1571.157} C_VEL
LIN {X 0,Y 587.337,Z 382.323,A -85,B 0,C 180,E1 -1574.114,E2 -1574.114} C_VEL
LIN {X 0,Y 587.314,Z 382.329,A -85,B 0,C 180,E1 -1576.993,E2 -1576.993} C_VEL
LIN {X 0,Y 587.319,Z 382.323,A -85,B 0,C 180,E1 -1579.746,E2 -1579.746} C_VEL
LIN {X 0,Y 587.346,Z 382.326,A -85,B 0,C 180,E1 -1582.392,E2 -1582.392} C_VEL
LIN {X 0,Y 587.33,Z 382.322,A -85,B 0,C 180,E1 -1584.944,E2 -1584.944} C_VEL
LIN {X 0,Y 587.341,Z 382.328,A -85,B 0,C 180,E1 -1587.421,E2 -1587.421} C_VEL
LIN {X 0,Y 587.336,Z 382.321,A -85,B 0,C 180,E1 -1589.83,E2 -1589.83} C_VEL
LIN {X 0,Y 587.354,Z 382.322,A -85,B 0,C 180,E1 -1592.307,E2 -1592.307} C_VEL
LIN {X 0,Y 587.338,Z 382.326,A -85,B 0,C 180,E1 -1594.483,E2 -1594.483} C_VEL
LIN {X 0,Y 587.339,Z 382.325,A -85,B 0,C 180,E1 -1597.486,E2 -1597.486} C_VEL
LIN {X 0,Y 587.346,Z 382.32,A -85,B 0,C 180,E1 -1600.425,E2 -1600.425} C_VEL
LIN {X 0,Y 587.353,Z 382.32,A -85,B 0,C 180,E1 -1603.311,E2 -1603.311} C_VEL
LIN {X 0,Y 587.364,Z 382.323,A -85,B 0,C 180,E1 -1606.154,E2 -1606.154} C_VEL
LIN {X 0,Y 587.342,Z 382.32,A -85,B 0,C 180,E1 -1608.962,E2 -1608.962} C_VEL
LIN {X 0,Y 587.37,Z 382.32,A -85,B 0,C 180,E1 -1611.745,E2 -1611.745} C_VEL
LIN {X 0,Y 587.358,Z 382.321,A -85,B 0,C 180,E1 -1614.507,E2 -1614.507} C_VEL
LIN {X 0,Y 587.376,Z 382.316,A -85,B 0,C 180,E1 -1617.257,E2 -1617.257} C_VEL
LIN {X 0,Y 587.386,Z 382.322,A -85,B 0,C 180,E1 -1620,E2 -1620} C_VEL
LIN {X 0,Y 587.376,Z 382.316,A -85,B 0,C 180,E1 -1622.743,E2 -1622.743} C_VEL
LIN {X 0,Y 587.361,Z 382.321,A -85,B 0,C 180,E1 -1625.493,E2 -1625.493} C_VEL
LIN {X 0,Y 587.371,Z 382.32,A -85,B 0,C 180,E1 -1628.255,E2 -1628.255} C_VEL
LIN {X 0,Y 587.351,Z 382.319,A -85,B 0,C 180,E1 -1631.134,E2 -1631.134} C_VEL
LIN {X 0,Y 587.368,Z 382.318,A -85,B 0,C 180,E1 -1634.26,E2 -1634.26} C_VEL
LIN {X 0,Y 587.347,Z 382.324,A -85,B 0,C 180,E1 -1637.406,E2 -1637.406} C_VEL
LIN {X 0,Y 587.306,Z 382.326,A -85,B 0,C 180,E1 -1638.313,E2 -1638.313} C_VEL
LIN {X 0,Y 586.666,Z 382.411,A -85,B 0,C 180,E1 -1638.885,E2 -1638.885} C_VEL
LIN {X 0,Y 583.844,Z 382.76,A -85,B 0,C 180,E1 -1639.814,E2 -1639.814} C_VEL
LIN {X 0,Y 581.434,Z 383.063,A -85,B 0,C 180,E1 -1640.561,E2 -1640.561} C_VEL
LIN {X 0,Y 580.38,Z 383.189,A -85,B 0,C 180,E1 -1641.137,E2 -1641.137} C_VEL
LIN {X 0,Y 580.286,Z 383.199,A -85,B 0,C 180,E1 -1641.332,E2 -1641.332} C_VEL
LIN {X 0,Y 580.301,Z 383.2,A -85,B 0,C 180,E1 -1644.316,E2 -1644.316} C_VEL
LIN {X 0,Y 580.282,Z 383.199,A -85,B 0,C 180,E1 -1646.623,E2 -1646.623} C_VEL
LIN {X 0,Y 580.304,Z 383.202,A -85,B 0,C 180,E1 -1649.31,E2 -1649.31} C_VEL
LIN {X 0,Y 580.299,Z 383.2,A -85,B 0,C 180,E1 -1652.201,E2 -1652.201} C_VEL
LIN {X 0,Y 580.303,Z 383.199,A -85,B 0,C 180,E1 -1654.696,E2 -1654.696} C_VEL
LIN {X 0,Y 580.303,Z 383.199,A -85,B 0,C 180,E1 -1657.268,E2 -1657.268} C_VEL
LIN {X 0,Y 580.299,Z 383.197,A -85,B 0,C 180,E1 -1660.271,E2 -1660.271} C_VEL
LIN {X 0,Y 580.279,Z 383.205,A -85,B 0,C 180,E1 -1662.706,E2 -1662.706} C_VEL
LIN {X 0,Y 580.278,Z 383.201,A -85,B 0,C 180,E1 -1665.609,E2 -1665.609} C_VEL
LIN {X 0,Y 580.317,Z 383.2,A -85,B 0,C 180,E1 -1668.234,E2 -1668.234} C_VEL
LIN {X 0,Y 580.28,Z 383.201,A -85,B 0,C 180,E1 -1670.965,E2 -1670.965} C_VEL
LIN {X 0,Y 580.265,Z 383.204,A -85,B 0,C 180,E1 -1673.596,E2 -1673.596} C_VEL
LIN {X 0,Y 580.219,Z 383.21,A -85,B 0,C 180,E1 -1674.45,E2 -1674.45} C_VEL
LIN {X 0,Y 580.284,Z 384.388,A -85,B 0,C 180,E1 -1675.444,E2 -1675.444} C_VEL
LIN {X 0,Y 580.24,Z 388.564,A -85,B 0,C 180,E1 -1677.98,E2 -1677.98} C_VEL
LIN {X 0,Y 580.204,Z 393.673,A -85,B 0,C 180,E1 -1681.019,E2 -1681.019} C_VEL
LIN {X 0,Y 580.16,Z 398.278,A -85,B 0,C 180,E1 -1683.693,E2 -1683.693} C_VEL
LIN {X 0,Y 580.136,Z 403.188,A -85,B 0,C 180,E1 -1686.436,E2 -1686.436} C_VEL
LIN {X 0,Y 580.132,Z 407.687,A -85,B 0,C 180,E1 -1688.879,E2 -1688.879} C_VEL
LIN {X 0,Y 580.109,Z 412.864,A -85,B 0,C 180,E1 -1691.64,E2 -1691.64} C_VEL
LIN {X 0,Y 580.096,Z 417.012,A -85,B 0,C 180,E1 -1693.82,E2 -1693.82} C_VEL
LIN {X 0,Y 580.1,Z 421.159,A -85,B 0,C 180,E1 -1695.978,E2 -1695.978} C_VEL
LIN {X 0,Y 580.081,Z 424.529,A -85,B 0,C 180,E1 -1697.715,E2 -1697.715} C_VEL
LIN {X 0,Y 580.798,Z 430.494,A -85,B 0,C 180,E1 -1697.863,E2 -1697.863} C_VEL
LIN {X 0,Y 580.696,Z 443.155,A -85,B 0,C 180,E1 -1698.216,E2 -1698.216} C_VEL
LIN {X 0,Y 580.618,Z 455.275,A -85,B 0,C 180,E1 -1698.692,E2 -1698.692} C_VEL
LIN {X 0,Y 580.538,Z 466.549,A -85,B 0,C 180,E1 -1699.273,E2 -1699.273} C_VEL
LIN {X 0,Y 580.452,Z 477.329,A -85,B 0,C 180,E1 -1699.977,E2 -1699.977} C_VEL
LIN {X 0,Y 580.333,Z 487.104,A -85,B 0,C 180,E1 -1700.766,E2 -1700.766} C_VEL
LIN {X 0,Y 580.264,Z 495.996,A -85,B 0,C 180,E1 -1701.643,E2 -1701.643} C_VEL
LIN {X 0,Y 580.205,Z 504.68,A -85,B 0,C 180,E1 -1702.693,E2 -1702.693} C_VEL
LIN {X 0,Y 580.137,Z 511.607,A -85,B 0,C 180,E1 -1703.741,E2 -1703.741} C_VEL
LIN {X 0,Y 580.085,Z 517.157,A -85,B 0,C 180,E1 -1704.787,E2 -1704.787} C_VEL
LIN {X 0,Y 580.105,Z 521.518,A -85,B 0,C 180,E1 -1705.832,E2 -1705.832} C_VEL
LIN {X 0,Y 580.123,Z 523.821,A -85,B 0,C 180,E1 -1706.527,E2 -1706.527} C_VEL
LIN {X 0,Y 580.043,Z 525.698,A -85,B 0,C 180,E1 -1707.222,E2 -1707.222} C_VEL
LIN {X 0,Y 580.04,Z 527.128,A -85,B 0,C 180,E1 -1707.917,E2 -1707.917} C_VEL
LIN {X 0,Y 580.04,Z 528.755,A -85,B 0,C 180,E1 -1709.306,E2 -1709.306} C_VEL
LIN {X 0,Y 580.038,Z 528.996,A -85,B 0,C 180,E1 -1710,E2 -1710} C_VEL
LIN {X 0,Y 580.04,Z 528.815,A -85,B 0,C 180,E1 -1710.694,E2 -1710.694} C_VEL
LIN {X 0,Y 580.04,Z 527.272,A -85,B 0,C 180,E1 -1712.083,E2 -1712.083} C_VEL
LIN {X 0,Y 580.044,Z 525.911,A -85,B 0,C 180,E1 -1712.778,E2 -1712.778} C_VEL
LIN {X 0,Y 580.11,Z 523.034,A -85,B 0,C 180,E1 -1713.821,E2 -1713.821} C_VEL
LIN {X 0,Y 580.053,Z 519.133,A -85,B 0,C 180,E1 -1714.865,E2 -1714.865} C_VEL
LIN {X 0,Y 580.162,Z 514.101,A -85,B 0,C 180,E1 -1715.91,E2 -1715.91} C_VEL
LIN {X 0,Y 580.158,Z 507.779,A -85,B 0,C 180,E1 -1716.958,E2 -1716.958} C_VEL
LIN {X 0,Y 580.241,Z 499.859,A -85,B 0,C 180,E1 -1718.007,E2 -1718.007} C_VEL
LIN {X 0,Y 580.308,Z 490.01,A -85,B 0,C 180,E1 -1719.058,E2 -1719.058} C_VEL
LIN {X 0,Y 580.421,Z 479.689,A -85,B 0,C 180,E1 -1719.936,E2 -1719.936} C_VEL
LIN {X 0,Y 580.524,Z 468.056,A -85,B 0,C 180,E1 -1720.727,E2 -1720.727} C_VEL
LIN {X 0,Y 580.63,Z 456.291,A -85,B 0,C 180,E1 -1721.352,E2 -1721.352} C_VEL
LIN {X 0,Y 580.68,Z 444.621,A -85,B 0,C 180,E1 -1721.825,E2 -1721.825} C_VEL
LIN {X 0,Y 580.782,Z 431.461,A -85,B 0,C 180,E1 -1722.204,E2 -1722.204} C_VEL
LIN {X 0,Y 580.479,Z 427.255,A -85,B 0,C 180,E1 -1722.299,E2 -1722.299} C_VEL
LIN {X 0,Y 580.096,Z 424.531,A -85,B 0,C 180,E1 -1722.374,E2 -1722.374} C_VEL
LIN {X 0,Y 580.105,Z 419.95,A -85,B 0,C 180,E1 -1724.739,E2 -1724.739} C_VEL
LIN {X 0,Y 580.083,Z 414.417,A -85,B 0,C 180,E1 -1727.631,E2 -1727.631} C_VEL
LIN {X 0,Y 580.099,Z 410.268,A -85,B 0,C 180,E1 -1729.83,E2 -1729.83} C_VEL
LIN {X 0,Y 580.129,Z 406.118,A -85,B 0,C 180,E1 -1732.059,E2 -1732.059} C_VEL
LIN {X 0,Y 580.157,Z 400.586,A -85,B 0,C 180,E1 -1735.087,E2 -1735.087} C_VEL
LIN {X 0,Y 580.215,Z 395.775,A -85,B 0,C 180,E1 -1737.843,E2 -1737.843} C_VEL
LIN {X 0,Y 580.198,Z 390.964,A -85,B 0,C 180,E1 -1740.68,E2 -1740.68} C_VEL
LIN {X 0,Y 580.245,Z 386.57,A -85,B 0,C 180,E1 -1743.307,E2 -1743.307} C_VEL
LIN {X 0,Y 580.275,Z 384.304,A -85,B 0,C 180,E1 -1744.697,E2 -1744.697} C_VEL
LIN {X 0,Y 580.22,Z 383.211,A -85,B 0,C 180,E1 -1745.55,E2 -1745.55} C_VEL
LIN {X 0,Y 580.291,Z 383.199,A -85,B 0,C 180,E1 -1748.146,E2 -1748.146} C_VEL
LIN {X 0,Y 580.301,Z 383.199,A -85,B 0,C 180,E1 -1750.843,E2 -1750.843} C_VEL
LIN {X 0,Y 580.292,Z 383.204,A -85,B 0,C 180,E1 -1753.657,E2 -1753.657} C_VEL
LIN {X 0,Y 580.276,Z 383.201,A -85,B 0,C 180,E1 -1756.61,E2 -1756.61} C_VEL
LIN {X 0,Y 580.302,Z 383.201,A -85,B 0,C 180,E1 -1759.157,E2 -1759.157} C_VEL
LIN {X 0,Y 580.293,Z 383.2,A -85,B 0,C 180,E1 -1761.927,E2 -1761.927} C_VEL
LIN {X 0,Y 580.256,Z 383.205,A -85,B 0,C 180,E1 -1764.453,E2 -1764.453} C_VEL
LIN {X 0,Y 580.293,Z 383.2,A -85,B 0,C 180,E1 -1766.975,E2 -1766.975} C_VEL
LIN {X 0,Y 580.3,Z 383.202,A -85,B 0,C 180,E1 -1769.425,E2 -1769.425} C_VEL
LIN {X 0,Y 580.301,Z 383.199,A -85,B 0,C 180,E1 -1772.141,E2 -1772.141} C_VEL
LIN {X 0,Y 580.326,Z 383.194,A -85,B 0,C 180,E1 -1775.27,E2 -1775.27} C_VEL
LIN {X 0,Y 580.276,Z 383.206,A -85,B 0,C 180,E1 -1777.947,E2 -1777.947} C_VEL
LIN {X 0,Y 580.304,Z 383.201,A -85,B 0,C 180,E1 -1780.913,E2 -1780.913} C_VEL
LIN {X 0,Y 580.28,Z 383.2,A -85,B 0,C 180,E1 -1783.826,E2 -1783.826} C_VEL
LIN {X 0,Y 580.329,Z 383.196,A -85,B 0,C 180,E1 -1785.983,E2 -1785.983} C_VEL
LIN {X 0,Y 580.309,Z 383.196,A -85,B 0,C 180,E1 -1788.827,E2 -1788.827} C_VEL
LIN {X 0,Y 580.336,Z 383.198,A -85,B 0,C 180,E1 -1791.644,E2 -1791.644} C_VEL
LIN {X 0,Y 580.327,Z 383.196,A -85,B 0,C 180,E1 -1794.44,E2 -1794.44} C_VEL
LIN {X 0,Y 580.342,Z 383.193,A -85,B 0,C 180,E1 -1797.223,E2 -1797.223} C_VEL
LIN {X 0,Y 580.354,Z 383.198,A -85,B 0,C 180,E1 -1800,E2 -1800} C_VEL
LIN {X 0,Y 580.343,Z 383.192,A -85,B 0,C 180,E1 -1802.776,E2 -1802.776} C_VEL
LIN {X 0,Y 580.324,Z 383.197,A -85,B 0,C 180,E1 -1805.56,E2 -1805.56} C_VEL
LIN {X 0,Y 580.336,Z 383.197,A -85,B 0,C 180,E1 -1808.356,E2 -1808.356} C_VEL
LIN {X 0,Y 580.304,Z 383.197,A -85,B 0,C 180,E1 -1811.191,E2 -1811.191} C_VEL
LIN {X 0,Y 580.331,Z 383.197,A -85,B 0,C 180,E1 -1814.017,E2 -1814.017} C_VEL
LIN {X 0,Y 580.316,Z 383.199,A -85,B 0,C 180,E1 -1816.914,E2 -1816.914} C_VEL
LIN {X 0,Y 580.309,Z 383.197,A -85,B 0,C 180,E1 -1819.822,E2 -1819.822} C_VEL
LIN {X 0,Y 580.294,Z 383.2,A -85,B 0,C 180,E1 -1822.803,E2 -1822.803} C_VEL
LIN {X 0,Y 580.31,Z 383.197,A -85,B 0,C 180,E1 -1825.08,E2 -1825.08} C_VEL
LIN {X 0,Y 580.301,Z 383.197,A -85,B 0,C 180,E1 -1828.186,E2 -1828.186} C_VEL
LIN {X 0,Y 580.288,Z 383.204,A -85,B 0,C 180,E1 -1830.695,E2 -1830.695} C_VEL
LIN {X 0,Y 580.306,Z 383.197,A -85,B 0,C 180,E1 -1833.316,E2 -1833.316} C_VEL
LIN {X 0,Y 580.265,Z 383.206,A -85,B 0,C 180,E1 -1835.758,E2 -1835.758} C_VEL
LIN {X 0,Y 580.291,Z 383.201,A -85,B 0,C 180,E1 -1838.146,E2 -1838.146} C_VEL
LIN {X 0,Y 580.302,Z 383.2,A -85,B 0,C 180,E1 -1840.843,E2 -1840.843} C_VEL
LIN {X 0,Y 580.282,Z 383.199,A -85,B 0,C 180,E1 -1843.658,E2 -1843.658} C_VEL
LIN {X 0,Y 580.289,Z 383.202,A -85,B 0,C 180,E1 -1846.608,E2 -1846.608} C_VEL
LIN {X 0,Y 580.301,Z 383.199,A -85,B 0,C 180,E1 -1849.157,E2 -1849.157} C_VEL
LIN {X 0,Y 580.292,Z 383.201,A -85,B 0,C 180,E1 -1851.927,E2 -1851.927} C_VEL
LIN {X 0,Y 580.319,Z 383.385,A -85,B 0,C 180,E1 -1853.94,E2 -1853.94} C_VEL
LIN {X 0,Y 580.522,Z 387.168,A -85,B 0,C 180,E1 -1855.41,E2 -1855.41} C_VEL
LIN {X 0,Y 580.485,Z 393.957,A -85,B 0,C 180,E1 -1857.941,E2 -1857.941} C_VEL
LIN {X 0,Y 580.434,Z 401.6,A -85,B 0,C 180,E1 -1860.668,E2 -1860.668} C_VEL
LIN {X 0,Y 580.356,Z 410.207,A -85,B 0,C 180,E1 -1863.654,E2 -1863.654} C_VEL
LIN {X 0,Y 580.302,Z 418.334,A -85,B 0,C 180,E1 -1866.443,E2 -1866.443} C_VEL
LIN {X 0,Y 580.245,Z 427.239,A -85,B 0,C 180,E1 -1869.436,E2 -1869.436} C_VEL
LIN {X 0,Y 580.205,Z 436.143,A -85,B 0,C 180,E1 -1872.373,E2 -1872.373} C_VEL
LIN {X 0,Y 580.147,Z 445.048,A -85,B 0,C 180,E1 -1875.262,E2 -1875.262} C_VEL
LIN {X 0,Y 580.132,Z 452.491,A -85,B 0,C 180,E1 -1877.649,E2 -1877.649} C_VEL
LIN {X 0,Y 580.808,Z 457.224,A -85,B 0,C 180,E1 -1877.752,E2 -1877.752} C_VEL
LIN {X 0,Y 580.73,Z 470.494,A -85,B 0,C 180,E1 -1878.083,E2 -1878.083} C_VEL
LIN {X 0,Y 580.629,Z 482.316,A -85,B 0,C 180,E1 -1878.515,E2 -1878.515} C_VEL
LIN {X 0,Y 580.561,Z 494.209,A -85,B 0,C 180,E1 -1879.097,E2 -1879.097} C_VEL
LIN {X 0,Y 580.452,Z 505.478,A -85,B 0,C 180,E1 -1879.8,E2 -1879.8} C_VEL
LIN {X 0,Y 580.352,Z 515.646,A -85,B 0,C 180,E1 -1880.591,E2 -1880.591} C_VEL
LIN {X 0,Y 580.279,Z 524.786,A -85,B 0,C 180,E1 -1881.468,E2 -1881.468} C_VEL
LIN {X 0,Y 580.199,Z 533.689,A -85,B 0,C 180,E1 -1882.518,E2 -1882.518} C_VEL
LIN {X 0,Y 580.12,Z 540.465,A -85,B 0,C 180,E1 -1883.505,E2 -1883.505} C_VEL
LIN {X 0,Y 580.139,Z 545.68,A -85,B 0,C 180,E1 -1884.438,E2 -1884.438} C_VEL
LIN {X 0,Y 580.108,Z 550.371,A -85,B 0,C 180,E1 -1885.483,E2 -1885.483} C_VEL
LIN {X 0,Y 580.123,Z 553.957,A -85,B 0,C 180,E1 -1886.527,E2 -1886.527} C_VEL
LIN {X 0,Y 580.043,Z 555.808,A -85,B 0,C 180,E1 -1887.222,E2 -1887.222} C_VEL
LIN {X 0,Y 580.04,Z 557.2,A -85,B 0,C 180,E1 -1887.917,E2 -1887.917} C_VEL
LIN {X 0,Y 580.04,Z 558.784,A -85,B 0,C 180,E1 -1889.306,E2 -1889.306} C_VEL
LIN {X 0,Y 580.037,Z 559,A -85,B 0,C 180,E1 -1890,E2 -1890} C_VEL
LIN {X 0,Y 580.047,Z 558.186,A -85,B 0,C 180,E1 -1891.388,E2 -1891.388} C_VEL
LIN {X 0,Y 580.04,Z 557.201,A -85,B 0,C 180,E1 -1892.083,E2 -1892.083} C_VEL
LIN {X 0,Y 580.043,Z 555.81,A -85,B 0,C 180,E1 -1892.778,E2 -1892.778} C_VEL
LIN {X 0,Y 580.109,Z 552.896,A -85,B 0,C 180,E1 -1893.821,E2 -1893.821} C_VEL
LIN {X 0,Y 580.054,Z 548.949,A -85,B 0,C 180,E1 -1894.865,E2 -1894.865} C_VEL
LIN {X 0,Y 580.139,Z 542.878,A -85,B 0,C 180,E1 -1896.085,E2 -1896.085} C_VEL
LIN {X 0,Y 580.184,Z 536.237,A -85,B 0,C 180,E1 -1897.132,E2 -1897.132} C_VEL
LIN {X 0,Y 580.25,Z 527.99,A -85,B 0,C 180,E1 -1898.182,E2 -1898.182} C_VEL
LIN {X 0,Y 580.308,Z 519.538,A -85,B 0,C 180,E1 -1899.058,E2 -1899.058} C_VEL
LIN {X 0,Y 580.425,Z 509.096,A -85,B 0,C 180,E1 -1899.936,E2 -1899.936} C_VEL
LIN {X 0,Y 580.491,Z 498.758,A -85,B 0,C 180,E1 -1900.64,E2 -1900.64} C_VEL
LIN {X 0,Y 580.596,Z 487.247,A -85,B 0,C 180,E1 -1901.264,E2 -1901.264} C_VEL
LIN {X 0,Y 580.671,Z 474.472,A -85,B 0,C 180,E1 -1901.785,E2 -1901.785} C_VEL
LIN {X 0,Y 580.77,Z 461.436,A -85,B 0,C 180,E1 -1902.16,E2 -1902.16} C_VEL
LIN {X 0,Y 580.565,Z 455.375,A -85,B 0,C 180,E1 -1902.289,E2 -1902.289} C_VEL
LIN {X 0,Y 580.131,Z 452.492,A -85,B 0,C 180,E1 -1902.351,E2 -1902.351} C_VEL
LIN {X 0,Y 580.158,Z 443.935,A -85,B 0,C 180,E1 -1905.097,E2 -1905.097} C_VEL
LIN {X 0,Y 580.208,Z 435.031,A -85,B 0,C 180,E1 -1907.992,E2 -1907.992} C_VEL
LIN {X 0,Y 580.245,Z 427.239,A -85,B 0,C 180,E1 -1910.564,E2 -1910.564} C_VEL
LIN {X 0,Y 580.301,Z 418.335,A -85,B 0,C 180,E1 -1913.557,E2 -1913.557} C_VEL
LIN {X 0,Y 580.356,Z 410.207,A -85,B 0,C 180,E1 -1916.346,E2 -1916.346} C_VEL
LIN {X 0,Y 580.434,Z 401.601,A -85,B 0,C 180,E1 -1919.332,E2 -1919.332} C_VEL
LIN {X 0,Y 580.49,Z 393.599,A -85,B 0,C 180,E1 -1922.189,E2 -1922.189} C_VEL
LIN {X 0,Y 580.553,Z 385.833,A -85,B 0,C 180,E1 -1925.101,E2 -1925.101} C_VEL
LIN {X 0,Y 580.288,Z 383.205,A -85,B 0,C 180,E1 -1926.147,E2 -1926.147} C_VEL
LIN {X 0,Y 580.297,Z 383.199,A -85,B 0,C 180,E1 -1929.185,E2 -1929.185} C_VEL
LIN {X 0,Y 580.317,Z 383.2,A -85,B 0,C 180,E1 -1931.766,E2 -1931.766} C_VEL
LIN {X 0,Y 580.272,Z 383.201,A -85,B 0,C 180,E1 -1934.626,E2 -1934.626} C_VEL
LIN {X 0,Y 580.288,Z 383.2,A -85,B 0,C 180,E1 -1937.628,E2 -1937.628} C_VEL
LIN {X 0,Y 580.296,Z 383.199,A -85,B 0,C 180,E1 -1940.067,E2 -1940.067} C_VEL
LIN {X 0,Y 580.304,Z 383.197,A -85,B 0,C 180,E1 -1943.065,E2 -1943.065} C_VEL
LIN {X 0,Y 580.299,Z 383.201,A -85,B 0,C 180,E1 -1945.442,E2 -1945.442} C_VEL
LIN {X 0,Y 580.305,Z 383.198,A -85,B 0,C 180,E1 -1947.969,E2 -1947.969} C_VEL
LIN {X 0,Y 580.303,Z 383.202,A -85,B 0,C 180,E1 -1950.69,E2 -1950.69} C_VEL
LIN {X 0,Y 580.295,Z 383.198,A -85,B 0,C 180,E1 -1953.666,E2 -1953.666} C_VEL
LIN {X 0,Y 580.301,Z 383.2,A -85,B 0,C 180,E1 -1955.684,E2 -1955.684} C_VEL
LIN {X 0,Y 580.287,Z 383.199,A -85,B 0,C 180,E1 -1958.695,E2 -1958.695} C_VEL
LIN {X 0,Y 580.322,Z 383.199,A -85,B 0,C 180,E1 -1960.914,E2 -1960.914} C_VEL
LIN {X 0,Y 580.281,Z 383.199,A -85,B 0,C 180,E1 -1963.826,E2 -1963.826} C_VEL
LIN {X 0,Y 580.33,Z 383.196,A -85,B 0,C 180,E1 -1965.983,E2 -1965.983} C_VEL
LIN {X 0,Y 580.308,Z 383.197,A -85,B 0,C 180,E1 -1968.827,E2 -1968.827} C_VEL
LIN {X 0,Y 580.335,Z 383.198,A -85,B 0,C 180,E1 -1971.644,E2 -1971.644} C_VEL
LIN {X 0,Y 580.324,Z 383.197,A -85,B 0,C 180,E1 -1974.44,E2 -1974.44} C_VEL
LIN {X 0,Y 580.342,Z 383.192,A -85,B 0,C 180,E1 -1977.224,E2 -1977.224} C_VEL
LIN {X 0,Y 580.355,Z 383.198,A -85,B 0,C 180,E1 -1980,E2 -1980} C_VEL
LIN {X 0,Y 580.342,Z 383.193,A -85,B 0,C 180,E1 -1982.777,E2 -1982.777} C_VEL
LIN {X 0,Y 580.327,Z 383.196,A -85,B 0,C 180,E1 -1985.56,E2 -1985.56} C_VEL
LIN {X 0,Y 580.336,Z 383.198,A -85,B 0,C 180,E1 -1988.356,E2 -1988.356} C_VEL
LIN {X 0,Y 580.303,Z 383.197,A -85,B 0,C 180,E1 -1991.191,E2 -1991.191} C_VEL
LIN {X 0,Y 580.329,Z 383.197,A -85,B 0,C 180,E1 -1994.017,E2 -1994.017} C_VEL
LIN {X 0,Y 580.315,Z 383.2,A -85,B 0,C 180,E1 -1996.914,E2 -1996.914} C_VEL
LIN {X 0,Y 580.308,Z 383.197,A -85,B 0,C 180,E1 -1999.822,E2 -1999.822} C_VEL
LIN {X 0,Y 580.286,Z 383.199,A -85,B 0,C 180,E1 -2001.332,E2 -2001.332} C_VEL
LIN {X 0,Y 579.588,Z 383.29,A -85,B 0,C 180,E1 -2001.912,E2 -2001.912} C_VEL
LIN {X 0,Y 576.71,Z 383.646,A -85,B 0,C 180,E1 -2002.851,E2 -2002.851} C_VEL
LIN {X 0,Y 574.315,Z 383.945,A -85,B 0,C 180,E1 -2003.608,E2 -2003.608} C_VEL
LIN {X 0,Y 573.318,Z 384.072,A -85,B 0,C 180,E1 -2004.192,E2 -2004.192} C_VEL
LIN {X 0,Y 573.252,Z 384.076,A -85,B 0,C 180,E1 -2004.389,E2 -2004.389} C_VEL
LIN {X 0,Y 573.255,Z 384.076,A -85,B 0,C 180,E1 -2006.976,E2 -2006.976} C_VEL
LIN {X 0,Y 573.249,Z 384.079,A -85,B 0,C 180,E1 -2009.488,E2 -2009.488} C_VEL
LIN {X 0,Y 573.255,Z 384.081,A -85,B 0,C 180,E1 -2012.645,E2 -2012.645} C_VEL
LIN {X 0,Y 573.271,Z 384.073,A -85,B 0,C 180,E1 -2015.184,E2 -2015.184} C_VEL
LIN {X 0,Y 573.239,Z 384.083,A -85,B 0,C 180,E1 -2017.808,E2 -2017.808} C_VEL
LIN {X 0,Y 573.273,Z 384.073,A -85,B 0,C 180,E1 -2020.528,E2 -2020.528} C_VEL
LIN {X 0,Y 573.241,Z 384.077,A -85,B 0,C 180,E1 -2023.668,E2 -2023.668} C_VEL
LIN {X 0,Y 573.25,Z 384.079,A -85,B 0,C 180,E1 -2026.642,E2 -2026.642} C_VEL
LIN {X 0,Y 573.247,Z 384.08,A -85,B 0,C 180,E1 -2029.475,E2 -2029.475} C_VEL
LIN {X 0,Y 573.238,Z 384.077,A -85,B 0,C 180,E1 -2032.193,E2 -2032.193} C_VEL
LIN {X 0,Y 573.155,Z 384.241,A -85,B 0,C 180,E1 -2034.808,E2 -2034.808} C_VEL
LIN {X 0,Y 573.176,Z 388.348,A -85,B 0,C 180,E1 -2037.35,E2 -2037.35} C_VEL
LIN {X 0,Y 573.127,Z 392.401,A -85,B 0,C 180,E1 -2039.817,E2 -2039.817} C_VEL
LIN {X 0,Y 573.157,Z 396.463,A -85,B 0,C 180,E1 -2042.228,E2 -2042.228} C_VEL
LIN {X 0,Y 573.105,Z 401.493,A -85,B 0,C 180,E1 -2045.158,E2 -2045.158} C_VEL
LIN {X 0,Y 573.043,Z 405.954,A -85,B 0,C 180,E1 -2047.654,E2 -2047.654} C_VEL
LIN {X 0,Y 573.017,Z 410.101,A -85,B 0,C 180,E1 -2049.915,E2 -2049.915} C_VEL
LIN {X 0,Y 573.009,Z 414.248,A -85,B 0,C 180,E1 -2052.144,E2 -2052.144} C_VEL
LIN {X 0,Y 573.002,Z 419.778,A -85,B 0,C 180,E1 -2055.074,E2 -2055.074} C_VEL
LIN {X 0,Y 573.015,Z 424.53,A -85,B 0,C 180,E1 -2057.561,E2 -2057.561} C_VEL
LIN {X 0,Y 573.863,Z 431.431,A -85,B 0,C 180,E1 -2057.737,E2 -2057.737} C_VEL
LIN {X 0,Y 573.741,Z 444.469,A -85,B 0,C 180,E1 -2058.115,E2 -2058.115} C_VEL
LIN {X 0,Y 573.651,Z 456.662,A -85,B 0,C 180,E1 -2058.615,E2 -2058.615} C_VEL
LIN {X 0,Y 573.545,Z 468.049,A -85,B 0,C 180,E1 -2059.231,E2 -2059.231} C_VEL
LIN {X 0,Y 573.405,Z 479.673,A -85,B 0,C 180,E1 -2060.031,E2 -2060.031} C_VEL
LIN {X 0,Y 573.287,Z 489.051,A -85,B 0,C 180,E1 -2060.83,E2 -2060.83} C_VEL
LIN {X 0,Y 573.201,Z 497.611,A -85,B 0,C 180,E1 -2061.717,E2 -2061.717} C_VEL
LIN {X 0,Y 573.138,Z 505.924,A -85,B 0,C 180,E1 -2062.78,E2 -2062.78} C_VEL
LIN {X 0,Y 573.065,Z 512.621,A -85,B 0,C 180,E1 -2063.84,E2 -2063.84} C_VEL
LIN {X 0,Y 572.962,Z 518.763,A -85,B 0,C 180,E1 -2065.074,E2 -2065.074} C_VEL
LIN {X 0,Y 573.015,Z 522.752,A -85,B 0,C 180,E1 -2066.132,E2 -2066.132} C_VEL
LIN {X 0,Y 572.959,Z 525.7,A -85,B 0,C 180,E1 -2067.188,E2 -2067.188} C_VEL
LIN {X 0,Y 572.94,Z 527.128,A -85,B 0,C 180,E1 -2067.891,E2 -2067.891} C_VEL
LIN {X 0,Y 572.941,Z 528.755,A -85,B 0,C 180,E1 -2069.297,E2 -2069.297} C_VEL
LIN {X 0,Y 572.939,Z 528.996,A -85,B 0,C 180,E1 -2070,E2 -2070} C_VEL
LIN {X 0,Y 572.94,Z 528.815,A -85,B 0,C 180,E1 -2070.703,E2 -2070.703} C_VEL
LIN {X 0,Y 572.94,Z 527.27,A -85,B 0,C 180,E1 -2072.109,E2 -2072.109} C_VEL
LIN {X 0,Y 572.96,Z 525.909,A -85,B 0,C 180,E1 -2072.812,E2 -2072.812} C_VEL
LIN {X 0,Y 573.015,Z 523.032,A -85,B 0,C 180,E1 -2073.868,E2 -2073.868} C_VEL
LIN {X 0,Y 572.963,Z 519.131,A -85,B 0,C 180,E1 -2074.926,E2 -2074.926} C_VEL
LIN {X 0,Y 573.076,Z 514.099,A -85,B 0,C 180,E1 -2075.984,E2 -2075.984} C_VEL
LIN {X 0,Y 573.083,Z 507.775,A -85,B 0,C 180,E1 -2077.044,E2 -2077.044} C_VEL
LIN {X 0,Y 573.175,Z 499.854,A -85,B 0,C 180,E1 -2078.106,E2 -2078.106} C_VEL
LIN {X 0,Y 573.287,Z 490.004,A -85,B 0,C 180,E1 -2079.17,E2 -2079.17} C_VEL
LIN {X 0,Y 573.423,Z 479.683,A -85,B 0,C 180,E1 -2080.058,E2 -2080.058} C_VEL
LIN {X 0,Y 573.526,Z 468.095,A -85,B 0,C 180,E1 -2080.857,E2 -2080.857} C_VEL
LIN {X 0,Y 573.658,Z 457.198,A -85,B 0,C 180,E1 -2081.449,E2 -2081.449} C_VEL
LIN {X 0,Y 573.732,Z 444.605,A -85,B 0,C 180,E1 -2081.97,E2 -2081.97} C_VEL
LIN {X 0,Y 573.858,Z 431.438,A -85,B 0,C 180,E1 -2082.353,E2 -2082.353} C_VEL
LIN {X 0,Y 573.208,Z 426.083,A -85,B 0,C 180,E1 -2082.48,E2 -2082.48} C_VEL
LIN {X 0,Y 572.987,Z 424.53,A -85,B 0,C 180,E1 -2082.53,E2 -2082.53} C_VEL
LIN {X 0,Y 573.002,Z 419.949,A -85,B 0,C 180,E1 -2084.926,E2 -2084.926} C_VEL
LIN {X 0,Y 572.991,Z 414.416,A -85,B 0,C 180,E1 -2087.857,E2 -2087.857} C_VEL
LIN {X 0,Y 573.016,Z 410.267,A -85,B 0,C 180,E1 -2090.085,E2 -2090.085} C_VEL
LIN {X 0,Y 573.043,Z 406.117,A -85,B 0,C 180,E1 -2092.346,E2 -2092.346} C_VEL
LIN {X 0,Y 573.092,Z 400.657,A -85,B 0,C 180,E1 -2095.418,E2 -2095.418} C_VEL
LIN {X 0,Y 573.133,Z 396.229,A -85,B 0,C 180,E1 -2098.006,E2 -2098.006} C_VEL
LIN {X 0,Y 573.154,Z 391.202,A -85,B 0,C 180,E1 -2100.998,E2 -2100.998} C_VEL
LIN {X 0,Y 573.189,Z 387.09,A -85,B 0,C 180,E1 -2103.512,E2 -2103.512} C_VEL
LIN {X 0,Y 573.186,Z 384.385,A -85,B 0,C 180,E1 -2105.19,E2 -2105.19} C_VEL
LIN {X 0,Y 573.255,Z 384.079,A -85,B 0,C 180,E1 -2107.166,E2 -2107.166} C_VEL
LIN {X 0,Y 573.243,Z 384.077,A -85,B 0,C 180,E1 -2109.608,E2 -2109.608} C_VEL
LIN {X 0,Y 573.247,Z 384.077,A -85,B 0,C 180,E1 -2112.642,E2 -2112.642} C_VEL
LIN {X 0,Y 573.218,Z 384.085,A -85,B 0,C 180,E1 -2115.326,E2 -2115.326} C_VEL
LIN {X 0,Y 573.243,Z 384.079,A -85,B 0,C 180,E1 -2117.6,E2 -2117.6} C_VEL
LIN {X 0,Y 573.256,Z 384.081,A -85,B 0,C 180,E1 -2120.567,E2 -2120.567} C_VEL
LIN {X 0,Y 573.256,Z 384.075,A -85,B 0,C 180,E1 -2123.078,E2 -2123.078} C_VEL
LIN {X 0,Y 573.272,Z 384.079,A -85,B 0,C 180,E1 -2125.671,E2 -2125.671} C_VEL
LIN {X 0,Y 573.244,Z 384.077,A -85,B 0,C 180,E1 -2128.185,E2 -2128.185} C_VEL
LIN {X 0,Y 573.267,Z 384.077,A -85,B 0,C 180,E1 -2130.634,E2 -2130.634} C_VEL
LIN {X 0,Y 573.255,Z 384.077,A -85,B 0,C 180,E1 -2133.024,E2 -2133.024} C_VEL
LIN {X 0,Y 573.279,Z 384.072,A -85,B 0,C 180,E1 -2135.366,E2 -2135.366} C_VEL
LIN {X 0,Y 573.233,Z 384.078,A -85,B 0,C 180,E1 -2138.419,E2 -2138.419} C_VEL
LIN {X 0,Y 573.283,Z 384.074,A -85,B 0,C 180,E1 -2140.728,E2 -2140.728} C_VEL
LIN {X 0,Y 573.252,Z 384.076,A -85,B 0,C 180,E1 -2143.622,E2 -2143.622} C_VEL
LIN {X 0,Y 573.277,Z 384.073,A -85,B 0,C 180,E1 -2145.807,E2 -2145.807} C_VEL
LIN {X 0,Y 573.267,Z 384.073,A -85,B 0,C 180,E1 -2148.745,E2 -2148.745} C_VEL
LIN {X 0,Y 573.293,Z 384.077,A -85,B 0,C 180,E1 -2151.541,E2 -2151.541} C_VEL
LIN {X 0,Y 573.294,Z 384.072,A -85,B 0,C 180,E1 -2154.372,E2 -2154.372} C_VEL
LIN {X 0,Y 573.306,Z 384.071,A -85,B 0,C 180,E1 -2157.892,E2 -2157.892} C_VEL
LIN {X 0,Y 573.335,Z 384.065,A -85,B 0,C 180,E1 -2160.702,E2 -2160.702} C_VEL
LIN {X 0,Y 573.235,Z 384.085,A -85,B 0,C 180,E1 -2163.514,E2 -2163.514} C_VEL
LIN {X 0,Y 573.292,Z 384.072,A -85,B 0,C 180,E1 -2165.628,E2 -2165.628} C_VEL
LIN {X 0,Y 573.293,Z 384.076,A -85,B 0,C 180,E1 -2168.459,E2 -2168.459} C_VEL
LIN {X 0,Y 573.276,Z 384.073,A -85,B 0,C 180,E1 -2171.312,E2 -2171.312} C_VEL
LIN {X 0,Y 573.286,Z 384.071,A -85,B 0,C 180,E1 -2174.425,E2 -2174.425} C_VEL
LIN {X 0,Y 573.262,Z 384.08,A -85,B 0,C 180,E1 -2177.112,E2 -2177.112} C_VEL
LIN {X 0,Y 573.257,Z 384.076,A -85,B 0,C 180,E1 -2180.077,E2 -2180.077} C_VEL
LIN {X 0,Y 573.238,Z 384.077,A -85,B 0,C 180,E1 -2183.099,E2 -2183.099} C_VEL
LIN {X 0,Y 573.258,Z 384.078,A -85,B 0,C 180,E1 -2185.41,E2 -2185.41} C_VEL
LIN {X 0,Y 573.254,Z 384.075,A -85,B 0,C 180,E1 -2188.029,E2 -2188.029} C_VEL
LIN {X 0,Y 573.233,Z 384.085,A -85,B 0,C 180,E1 -2190.882,E2 -2190.882} C_VEL
LIN {X 0,Y 573.266,Z 384.074,A -85,B 0,C 180,E1 -2193.524,E2 -2193.524} C_VEL
LIN {X 0,Y 573.242,Z 384.083,A -85,B 0,C 180,E1 -2196.05,E2 -2196.05} C_VEL
LIN {X 0,Y 573.251,Z 384.076,A -85,B 0,C 180,E1 -2198.701,E2 -2198.701} C_VEL
LIN {X 0,Y 573.233,Z 384.08,A -85,B 0,C 180,E1 -2201.457,E2 -2201.457} C_VEL
LIN {X 0,Y 573.239,Z 384.081,A -85,B 0,C 180,E1 -2204.333,E2 -2204.333} C_VEL
LIN {X 0,Y 573.247,Z 384.077,A -85,B 0,C 180,E1 -2207.358,E2 -2207.358} C_VEL
LIN {X 0,Y 573.241,Z 384.078,A -85,B 0,C 180,E1 -2210.392,E2 -2210.392} C_VEL
LIN {X 0,Y 573.255,Z 384.083,A -85,B 0,C 180,E1 -2213.078,E2 -2213.078} C_VEL
LIN {X 0,Y 573.244,Z 384.122,A -85,B 0,C 180,E1 -2213.733,E2 -2213.733} C_VEL
LIN {X 0,Y 573.528,Z 387.795,A -85,B 0,C 180,E1 -2215.187,E2 -2215.187} C_VEL
LIN {X 0,Y 573.482,Z 394.51,A -85,B 0,C 180,E1 -2217.736,E2 -2217.736} C_VEL
LIN {X 0,Y 573.428,Z 402.549,A -85,B 0,C 180,E1 -2220.643,E2 -2220.643} C_VEL
LIN {X 0,Y 573.316,Z 410.647,A -85,B 0,C 180,E1 -2223.492,E2 -2223.492} C_VEL
LIN {X 0,Y 573.266,Z 418.334,A -85,B 0,C 180,E1 -2226.136,E2 -2226.136} C_VEL
LIN {X 0,Y 573.23,Z 425.887,A -85,B 0,C 180,E1 -2228.716,E2 -2228.716} C_VEL
LIN {X 0,Y 573.159,Z 433.917,A -85,B 0,C 180,E1 -2231.409,E2 -2231.409} C_VEL
LIN {X 0,Y 573.11,Z 442.822,A -85,B 0,C 180,E1 -2234.348,E2 -2234.348} C_VEL
LIN {X 0,Y 573.081,Z 452.283,A -85,B 0,C 180,E1 -2237.427,E2 -2237.427} C_VEL
LIN {X 0,Y 573.089,Z 452.491,A -85,B 0,C 180,E1 -2237.495,E2 -2237.495} C_VEL
LIN {X 0,Y 573.879,Z 459.504,A -85,B 0,C 180,E1 -2237.647,E2 -2237.647} C_VEL
LIN {X 0,Y 573.78,Z 471.873,A -85,B 0,C 180,E1 -2237.981,E2 -2237.981} C_VEL
LIN {X 0,Y 573.671,Z 484.281,A -85,B 0,C 180,E1 -2238.462,E2 -2238.462} C_VEL
LIN {X 0,Y 573.585,Z 495.78,A -85,B 0,C 180,E1 -2239.052,E2 -2239.052} C_VEL
LIN {X 0,Y 573.445,Z 506.745,A -85,B 0,C 180,E1 -2239.764,E2 -2239.764} C_VEL
LIN {X 0,Y 573.308,Z 515.646,A -85,B 0,C 180,E1 -2240.474,E2 -2240.474} C_VEL
LIN {X 0,Y 573.215,Z 524.786,A -85,B 0,C 180,E1 -2241.362,E2 -2241.362} C_VEL
LIN {X 0,Y 573.142,Z 533.689,A -85,B 0,C 180,E1 -2242.425,E2 -2242.425} C_VEL
LIN {X 0,Y 573.051,Z 540.404,A -85,B 0,C 180,E1 -2243.415,E2 -2243.415} C_VEL
LIN {X 0,Y 573.07,Z 545.68,A -85,B 0,C 180,E1 -2244.37,E2 -2244.37} C_VEL
LIN {X 0,Y 573.028,Z 550.372,A -85,B 0,C 180,E1 -2245.427,E2 -2245.427} C_VEL
LIN {X 0,Y 573.022,Z 553.957,A -85,B 0,C 180,E1 -2246.484,E2 -2246.484} C_VEL
LIN {X 0,Y 572.959,Z 555.808,A -85,B 0,C 180,E1 -2247.188,E2 -2247.188} C_VEL
LIN {X 0,Y 572.939,Z 557.199,A -85,B 0,C 180,E1 -2247.891,E2 -2247.891} C_VEL
LIN {X 0,Y 572.941,Z 558.785,A -85,B 0,C 180,E1 -2249.297,E2 -2249.297} C_VEL
LIN {X 0,Y 572.938,Z 559,A -85,B 0,C 180,E1 -2250,E2 -2250} C_VEL
LIN {X 0,Y 572.946,Z 558.186,A -85,B 0,C 180,E1 -2251.406,E2 -2251.406} C_VEL
LIN {X 0,Y 572.94,Z 557.2,A -85,B 0,C 180,E1 -2252.109,E2 -2252.109} C_VEL
LIN {X 0,Y 572.959,Z 555.81,A -85,B 0,C 180,E1 -2252.812,E2 -2252.812} C_VEL
LIN {X 0,Y 573.014,Z 552.896,A -85,B 0,C 180,E1 -2253.868,E2 -2253.868} C_VEL
LIN {X 0,Y 572.963,Z 548.949,A -85,B 0,C 180,E1 -2254.926,E2 -2254.926} C_VEL
LIN {X 0,Y 573.064,Z 542.877,A -85,B 0,C 180,E1 -2256.16,E2 -2256.16} C_VEL
LIN {X 0,Y 573.119,Z 536.238,A -85,B 0,C 180,E1 -2257.221,E2 -2257.221} C_VEL
LIN {X 0,Y 573.201,Z 527.991,A -85,B 0,C 180,E1 -2258.283,E2 -2258.283} C_VEL
LIN {X 0,Y 573.287,Z 519.539,A -85,B 0,C 180,E1 -2259.17,E2 -2259.17} C_VEL
LIN {X 0,Y 573.429,Z 509.098,A -85,B 0,C 180,E1 -2260.058,E2 -2260.058} C_VEL
LIN {X 0,Y 573.546,Z 497.434,A -85,B 0,C 180,E1 -2260.853,E2 -2260.853} C_VEL
LIN {X 0,Y 573.651,Z 486.303,A -85,B 0,C 180,E1 -2261.446,E2 -2261.446} C_VEL
LIN {X 0,Y 573.753,Z 473.174,A -85,B 0,C 180,E1 -2261.974,E2 -2261.974} C_VEL
LIN {X 0,Y 573.869,Z 460.521,A -85,B 0,C 180,E1 -2262.331,E2 -2262.331} C_VEL
LIN {X 0,Y 573.481,Z 455.375,A -85,B 0,C 180,E1 -2262.443,E2 -2262.443} C_VEL
LIN {X 0,Y 573.089,Z 452.492,A -85,B 0,C 180,E1 -2262.505,E2 -2262.505} C_VEL
LIN {X 0,Y 573.087,Z 443.935,A -85,B 0,C 180,E1 -2265.288,E2 -2265.288} C_VEL
LIN {X 0,Y 573.147,Z 436.144,A -85,B 0,C 180,E1 -2267.852,E2 -2267.852} C_VEL
LIN {X 0,Y 573.201,Z 428.352,A -85,B 0,C 180,E1 -2270.453,E2 -2270.453} C_VEL
LIN {X 0,Y 573.249,Z 419.449,A -85,B 0,C 180,E1 -2273.481,E2 -2273.481} C_VEL
LIN {X 0,Y 573.316,Z 411.576,A -85,B 0,C 180,E1 -2276.187,E2 -2276.187} C_VEL
LIN {X 0,Y 573.392,Z 403.674,A -85,B 0,C 180,E1 -2278.957,E2 -2278.957} C_VEL
LIN {X 0,Y 573.449,Z 395.777,A -85,B 0,C 180,E1 -2281.803,E2 -2281.803} C_VEL
LIN {X 0,Y 573.519,Z 389.096,A -85,B 0,C 180,E1 -2284.311,E2 -2284.311} C_VEL
LIN {X 0,Y 573.526,Z 385.83,A -85,B 0,C 180,E1 -2285.576,E2 -2285.576} C_VEL
LIN {X 0,Y 573.238,Z 384.084,A -85,B 0,C 180,E1 -2286.322,E2 -2286.322} C_VEL
LIN {X 0,Y 573.243,Z 384.084,A -85,B 0,C 180,E1 -2288.702,E2 -2288.702} C_VEL
LIN {X 0,Y 573.256,Z 384.077,A -85,B 0,C 180,E1 -2291.595,E2 -2291.595} C_VEL
LIN {X 0,Y 573.242,Z 384.077,A -85,B 0,C 180,E1 -2294.333,E2 -2294.333} C_VEL
LIN {X 0,Y 573.242,Z 384.081,A -85,B 0,C 180,E1 -2297.359,E2 -2297.359} C_VEL
LIN {X 0,Y 573.25,Z 384.08,A -85,B 0,C 180,E1 -2300.393,E2 -2300.393} C_VEL
LIN {X 0,Y 573.258,Z 384.075,A -85,B 0,C 180,E1 -2303.078,E2 -2303.078} C_VEL
LIN {X 0,Y 573.271,Z 384.08,A -85,B 0,C 180,E1 -2305.671,E2 -2305.671} C_VEL
LIN {X 0,Y 573.243,Z 384.077,A -85,B 0,C 180,E1 -2308.185,E2 -2308.185} C_VEL
LIN {X 0,Y 573.266,Z 384.078,A -85,B 0,C 180,E1 -2310.634,E2 -2310.634} C_VEL
LIN {X 0,Y 573.255,Z 384.077,A -85,B 0,C 180,E1 -2313.024,E2 -2313.024} C_VEL
LIN {X 0,Y 573.277,Z 384.073,A -85,B 0,C 180,E1 -2315.366,E2 -2315.366} C_VEL
LIN {X 0,Y 573.23,Z 384.079,A -85,B 0,C 180,E1 -2318.419,E2 -2318.419} C_VEL
LIN {X 0,Y 573.281,Z 384.074,A -85,B 0,C 180,E1 -2320.728,E2 -2320.728} C_VEL
LIN {X 0,Y 573.253,Z 384.075,A -85,B 0,C 180,E1 -2323.622,E2 -2323.622} C_VEL
LIN {X 0,Y 573.277,Z 384.073,A -85,B 0,C 180,E1 -2325.807,E2 -2325.807} C_VEL
LIN {X 0,Y 573.265,Z 384.074,A -85,B 0,C 180,E1 -2328.745,E2 -2328.745} C_VEL
LIN {X 0,Y 573.291,Z 384.077,A -85,B 0,C 180,E1 -2331.541,E2 -2331.541} C_VEL
